// TwinCAT 3 PLC project lfe_motion
// Title: lcls-plc-lfe-motion
// Company: SLAC - LCLS
// ProjectVersion: 0.0.0
// ProgramVersion: 3.1.4026.17
// CompilerDefines: L
// libraries:
//   LCLS General, * (SLAC)
//   lcls-twincat-common-components, * (SLAC)
//   lcls-twincat-motion, * (SLAC)
//   lcls-twincat-physics, * (SLAC)
//   PMPS, * (SLAC - LCLS)
//   Tc2_MC2, * (Beckhoff Automation GmbH)
//   Tc2_SerialCom, * (Beckhoff Automation GmbH)
//   Tc2_Standard, * (Beckhoff Automation GmbH)
//   Tc2_System, * (Beckhoff Automation GmbH)
//   Tc3_Module, * (Beckhoff Automation GmbH)
// project tree:
//   DUTs/ DUT_SATT_Filter.TcDUT (not stored), ST_MPA.TcDUT (not stored), E_PositionState.TcDUT (not stored)
//   GVLs/ GVL.TcGVL, Main.TcGVL, RTDSL0.TcGVL (not stored)
//   / PlcTask.TcTTO
//   POUs/ FB_AttenuatorElementDensity.TcPOU (not stored), PRG_AL1L0_REF.TcPOU, PRG_IM5L0_PPM.TcPOU, PRG_3_PMPS_POST.TcPOU, PRG_4_LOG.TcPOU (not stored), PRG_AT2L0_SOLID.TcPOU, PRG_EM3L0_IPM.TcPOU, PRG_IM1L0_XTES.TcPOU, PRG_IM1L1_PPM.TcPOU (not stored), PRG_IM2L0_XTES.TcPOU, PRG_IM3L0_PPM.TcPOU, PRG_IM4L0_XTES.TcPOU, PRG_2_PMPS_PRE.TcPOU (not stored), PRG_1_PlcTask.TcPOU, PRG_RTDSL0.TcPOU (not stored), PRG_SL1L0_POWER.TcPOU (not stored), PRG_SL2L0_POWER.TcPOU (not stored), PRG_SL3L0_SCATTER.TcPOU, PRG_SP1L0_KMONO.TcPOU (not stored), PRG_PF1L0_WFS.TcPOU
//   Temp/ FB_AttFFO.TcPOU (not stored), FB_BasicAxisFFO.TcPOU (not stored), FB_BasicMotionStageAltFFO.TcPOU (not stored), FB_BasicMotionStageFFO.TcPOU (not stored), FB_MPA.TcPOU (not stored), FB_SimMotor.TcPOU (not stored), FB_SLITS.TcPOU (not stored), FB_SLITS_POWER.TcPOU (not stored), FB_SLITS_SCATTER.TcPOU
//   Version/ Global_Version.TcGVL
// real-time tasks:
//   TASK PlcTask: cycle T#10ms, priority 20, ADS port 350
// motion (NC):
//   TASK NC-Task 1 SAF: cycle T#1ms, priority 4, ADS port 501
//   TASK NC-Task 1 SVB: cycle T#10ms, priority 8, ADS port 511
//   AXIS Axis 1 (id 1)
//   AXIS Axis 2 (id 2)
//   AXIS Axis 3 (id 3)
//   AXIS Axis 4 (id 4)
//   AXIS Axis 5 (id 5)
//   AXIS Axis 6 (id 6)
//   AXIS Axis 7 (id 7)
//   AXIS Axis 8 (id 8)
//   AXIS Axis 9 (id 9)
//   AXIS Axis 10 (id 10)
//   AXIS Axis 11 (id 11)
//   AXIS Axis 12 (id 12)
//   AXIS Axis 13 (id 13)
//   AXIS Axis 14 (id 14)
//   AXIS Axis 15 (id 15)
//   AXIS Axis 16 (id 16)
//   AXIS Axis 17 (id 17)
//   AXIS Axis 18 (id 18)
//   AXIS Axis 19 (id 19)
//   AXIS Axis 20 IM1L0-XTES-MMS (id 20)
//   AXIS Axis 21 IM1L0-XTES-CLZ (id 21)
//   AXIS Axis 22 IM1L0-XTES-CLF (id 22)
//   AXIS Axis 23 IM1L1-PPM-MMS (id 23)
//   AXIS Axis 24 IM2L0-XTES-MMS (id 24)
//   AXIS Axis 25 IM2L0-XTES-CLZ (id 25)
//   AXIS Axis 26 IM2L0-XTES-CLF (id 26)
//   AXIS Axis 27 IM3L0-PPM-MMS (id 27)
//   AXIS Axis 28 IM4L0-XTES-MMS (id 28)
//   AXIS Axis 29 IM4L0-XTES-CLZ (id 29)
//   AXIS Axis 30 IM4L0-XTES-CLF (id 30)
//   AXIS PF1L0-WFS-MMS-01 (id 31)
//   AXIS PF1L0-WFS-MMS-02 (id 32)
//   AXIS Axis 33 (id 33)
//   AXIS Axis 34 (id 34)
//   AXIS Axis 35 (id 35)
//   AXIS Axis 36 (id 36)
//   AXIS Axis 37 (id 37)
//   AXIS Axis 38 (id 38)
//   AXIS Axis 39 (id 39)
//   AXIS Axis 40 (id 40)
//   AXIS SL1L0-BOTTOM-M41 (id 41)
//   AXIS SL1L0-SOUTH-M42 (id 42)
//   AXIS SL1L0-TOP-M43 (id 43)
//   AXIS SL1L0-NORTH-M44 (id 44)
//   AXIS SL2L0-BOTTOM-M45 (id 45)
//   AXIS SL2L0-SOUTH-M46 (id 46)
//   AXIS SL2L0-TOP-M47 (id 47)
//   AXIS SL2L0-NORTH-M48 (id 48)
//   AXIS XTAL ANGLE X (id 49)
//   AXIS XTAL VERT Y (id 50)
//   AXIS RETICLE HORIZ X (id 51)
//   AXIS RETICLE VERT Y (id 52)
//   AXIS DIODE HORIZ X (id 53)
//   AXIS DIODE VERT Y (id 54)
//   AXIS EM3L0-X-M55 (id 55)
//     Dynamic: AccelerationMaximum=50, DecelerationMaximum=50, Acceleration=50, Deceleration=50
//     Velo: RefSearch=0.1, RefSync=0.1, SlowManual=0.025, FastManual=0.05, Maximum=0.5
//     PositionAreaControl: Range=1
//     TargetPosControl: Range=0.001
//     OtherSettings: AllowMotionCmdToSlave=true
//     encoder EncType=29
//       EncPara: ScaleFactorNumerator=5e-05, Offset=-20.2296, MaxCount=#xffffffff, MaxCountHighDWord=#x0000001f
//         SoftEndMinControl: Enable=true, Range=-4
//         SoftEndMaxControl: Enable=true, Range=4
//         Inc: RefSoftSyncMask=#x0000ffff
//     drive DrvType=24
//       Analog: VeloReferenz=3.969, TorqueSetpointScale=10, ScaleFactorActTorque=0.1
//       TimeComp: TaskDelayCycles=1
//     controller CtrType=1
//       CtrPara: PriorControlFactor=1
//         PosDiffControl: Range=0.1
//         Observer: BandWidth=20
//   AXIS EM3L0-Y-M56 (id 56)
//     Dynamic: AccelerationMaximum=50, DecelerationMaximum=50, Acceleration=50, Deceleration=50
//     Velo: RefSearch=0.1, RefSync=0.1, SlowManual=0.025, FastManual=0.05, Maximum=2
//     PositionAreaControl: Enable=false
//     TargetPosControl: Range=0.025
//     OtherSettings: AllowMotionCmdToSlave=true
//     encoder EncType=29
//       EncPara: ScaleFactorNumerator=5e-05, Offset=3.65, Inverse=true, MaxCount=#xffffffff, MaxCountHighDWord=#x0000001f
//         SoftEndMinControl: Enable=true, Range=-81
//         SoftEndMaxControl: Enable=true, Range=1
//         Inc: RefSoftSyncMask=#x0000ffff
//     drive DrvType=24
//       Analog: VeloReferenz=12.5, TorqueSetpointScale=10, ScaleFactorActTorque=0.1
//       TimeComp: TaskDelayCycles=1
//     controller CtrType=1
//       CtrPara: PriorControlFactor=1
//         PosDiffControl: Enable=false, Range=0.03
//         Observer: BandWidth=20
//   AXIS Axis 57 IM5L0-PPM-MMS (id 57)
//     Dynamic: AccelerationMaximum=100, DecelerationMaximum=100, Acceleration=100, Deceleration=100, Jerk=1000
//     Velo: RefSearch=0.2, RefSync=0.2, SlowManual=0.05, FastManual=0.1, Maximum=1
//     TargetPosControl: Range=0.05
//     OtherSettings: AllowMotionCmdToSlave=true
//     encoder EncType=29
//       EncPara: ScaleFactorNumerator=5e-05, Offset=-6871886.7728, MaxCount=#xffffffff, MaxCountHighDWord=#x0000001f
//         SoftEndMinControl: Enable=true, Range=-105
//         SoftEndMaxControl: Enable=true
//         Inc: RefSoftSyncMask=#x0000ffff
//     drive DrvType=24
//       Analog: VeloReferenz=25, TorqueSetpointScale=10, ScaleFactorActTorque=0.1
//       TimeComp: TaskDelayCycles=1
//     controller CtrType=1
//       CtrPara: PriorControlFactor=1
//         PosDiffControl: Enable=false, Range=0.06
//         Observer: BandWidth=20
//   AXIS AL1L0-REF-MMS-M58 (id 58)
//     Dynamic: AccelerationMaximum=100, DecelerationMaximum=100, Acceleration=100, Deceleration=100
//     Velo: RefSearch=0.2, RefSync=0.2, SlowManual=0.05, FastManual=0.1, Maximum=1
//     PositionAreaControl: Range=1
//     TargetPosControl: Range=0.02
//     OtherSettings: AllowMotionCmdToSlave=true
//     encoder EncType=29
//       EncPara: ScaleFactorNumerator=5e-05, Offset=13.7558, Inverse=true, MaxCount=#xffffffff, MaxCountHighDWord=#x0000001f
//         SoftEndMinControl: Enable=true, Range=-47
//         SoftEndMaxControl: Enable=true, Range=2
//         Inc: RefSoftSyncMask=#x0000ffff
//     drive DrvType=24
//       Analog: VeloReferenz=5, TorqueSetpointScale=10, ScaleFactorActTorque=0.1
//       TimeComp: TaskDelayCycles=1
//     controller CtrType=1
//       CtrPara: PriorControlFactor=1
//         PosDiffControl: Range=1
//         PID: PosKp=2
//         Observer: BandWidth=20
//   AXIS SL3L0-BOTTOM-M59 (id 59)
//     Dynamic: AccelerationMaximum=100, DecelerationMaximum=100, Acceleration=100, Deceleration=100
//     Velo: Maximum=1
//     PositionAreaControl: Range=0.2
//     TargetPosControl: Range=0.005, Time=0.1
//     OtherSettings: AllowMotionCmdToSlave=true
//     encoder EncType=29
//       EncPara: ScaleFactorNumerator=5e-06, MaxCount=#xffffffff, MaxCountHighDWord=#x0000001f
//         SoftEndMinControl: Enable=true, Range=5.25
//         SoftEndMaxControl: Enable=true, Range=36.7
//         Inc: RefSoftSyncMask=#x0000ffff
//     drive DrvType=24
//       Analog: VeloReferenz=2, TorqueSetpointScale=10, ScaleFactorActTorque=0.1
//       TimeComp: TaskDelayCycles=1
//     controller CtrType=1
//       CtrPara: PriorControlFactor=1
//         PosDiffControl: Range=0.5
//         PID: PosKp=2
//         Observer: BandWidth=20
//   AXIS SL3L0-TOP-M60 (id 60)
//     Dynamic: AccelerationMaximum=100, DecelerationMaximum=100, Acceleration=100, Deceleration=100
//     Velo: Maximum=1
//     PositionAreaControl: Range=0.2
//     TargetPosControl: Range=0.005
//     OtherSettings: AllowMotionCmdToSlave=true
//     encoder EncType=29
//       EncPara: ScaleFactorNumerator=5e-06, MaxCount=#xffffffff, MaxCountHighDWord=#x0000001f
//         SoftEndMinControl: Enable=true, Range=4.5
//         SoftEndMaxControl: Enable=true, Range=33.3
//         Inc: RefSoftSyncMask=#x0000ffff
//     drive DrvType=24
//       Analog: VeloReferenz=2, TorqueSetpointScale=10, ScaleFactorActTorque=0.1
//       TimeComp: TaskDelayCycles=1
//     controller CtrType=1
//       CtrPara: PriorControlFactor=1
//         PosDiffControl: Range=0.5
//         PID: PosKp=2
//         Observer: BandWidth=20
//   AXIS SL3L0-SOUTH-M61 (id 61)
//     Dynamic: AccelerationMaximum=100, DecelerationMaximum=100, Acceleration=100, Deceleration=100
//     Velo: Maximum=1
//     PositionAreaControl: Range=0.2
//     TargetPosControl: Range=0.005
//     OtherSettings: AllowMotionCmdToSlave=true
//     encoder EncType=29
//       EncPara: ScaleFactorNumerator=5e-06, MaxCount=#xffffffff, MaxCountHighDWord=#x0000001f
//         SoftEndMinControl: Enable=true, Range=5
//         SoftEndMaxControl: Enable=true, Range=36.5
//         Inc: RefSoftSyncMask=#x0000ffff
//     drive DrvType=24
//       Analog: VeloReferenz=2, TorqueSetpointScale=10, ScaleFactorActTorque=0.1
//       TimeComp: TaskDelayCycles=1
//     controller CtrType=1
//       CtrPara: PriorControlFactor=1
//         PosDiffControl: Range=0.5
//         PID: PosKp=2
//         Observer: BandWidth=20
//   AXIS SL3L0-NORTH-M62 (id 62)
//     Dynamic: AccelerationMaximum=100, DecelerationMaximum=100, Acceleration=100, Deceleration=100
//     Velo: Maximum=1
//     PositionAreaControl: Range=0.2
//     TargetPosControl: Range=0.005
//     OtherSettings: AllowMotionCmdToSlave=true
//     encoder EncType=29
//       EncPara: ScaleFactorNumerator=5e-06, MaxCount=#xffffffff, MaxCountHighDWord=#x0000001f
//         SoftEndMinControl: Enable=true, Range=4.3
//         SoftEndMaxControl: Enable=true, Range=35.2
//         Inc: RefSoftSyncMask=#x0000ffff
//     drive DrvType=24
//       Analog: VeloReferenz=2, TorqueSetpointScale=10, ScaleFactorActTorque=0.1
//       TimeComp: TaskDelayCycles=1
//     controller CtrType=1
//       CtrPara: PriorControlFactor=1
//         PosDiffControl: Range=0.5
//         PID: PosKp=2
//         Observer: BandWidth=20
// I/O:
//   DEVICE PLC Rail (EtherCAT), AmsNetId 172.21.88.228.2.1
//     Power (EK1200) [EK1200-5000 EtherCAT Power supply (2A E-Bus)]
//       PMPS_FFO
//       License (EL6070)
//       PMPS_PRE
//       PLC Junction 1 (EK1122)
//       PLC Junction 2 (EK1122) [EK1122 2 port EtherCAT junction]
//         IM2L0 AT2L0 SL1L0 JUNCTION (CU1124)
//         X2 HXR EC2 (EK1100)
//         X2 SL2L0-Power (EK1100)
//       PLC Junction 3  (EK1122) [EK1122 2 port EtherCAT junction]
//         X1 B950-100H2-L0S5-ECJ-01 [CU1128 6x EtherCAT junction]
//           IM5L0-PPM [EK1100 EtherCAT Coupler (2A E-Bus)]
//             IM5L0-EL7047-E1 [EL7047 1Ch. Stepper motor output stage (50V, 5A)]
//             IM5L0-EL5042-E2 [EL5042 2Ch. BiSS-C Encoder]
//             IM5L0-EL2004-E3 [EL2004 4Ch. Dig. Output 24V, 0.5A]
//             IM5L0-EL1084-E4 [EL1084 4Ch. Dig. Input 24V, 3ms, negative]
//             IM5L0-EL3202-0010-E5 [EL3202-0010 2Ch. Ana. Input PT100 (RTD), High Precision]
//             IM5L0-EL3602-E6 [EL3602 2Ch. Ana. Input +/-10Volt, Diff. 24bit]
//             IM5L0-EL4004-E7 [EL4004 4Ch. Ana. Output 0-10V, 12bit]
//             IM5L0-EL2612-E8 [EL2612 2Ch. Relay Output, CO (125V AC / 30V DC)]
//             IM5L0-EL9011-E9 [EL9011 End Terminal]
//           SL3L0-SCATTER [EK1100 EtherCAT Coupler (2A E-Bus)]
//             SL3L0-EL7037-E1 [EL7037 1Ch. Stepper motor output stage (24V, 1.5A)]
//             SL3L0-EL5042-E2 [EL5042 2Ch. BiSS-C Encoder]
//             SL3L0-EL7037-E3 [EL7037 1Ch. Stepper motor output stage (24V, 1.5A)]
//             SL3L0-EL7037-E4 [EL7037 1Ch. Stepper motor output stage (24V, 1.5A)]
//             SL3L0-EL5042-E5 [EL5042 2Ch. BiSS-C Encoder]
//             SL3L0-EL7037-E6 [EL7037 1Ch. Stepper motor output stage (24V, 1.5A)]
//             SL3L0-EL9011-E7 [EL9011 End Terminal]
//           B950-100H2-L0S5-ECJ-01 (CU1128-B) [CU1128 6x EtherCAT junction - Dev A]
//             AL1L0-REF
//           B950-100H2-L0S5-ECJ-01 (CU1128-C) [CU1128 6x EtherCAT junction - Dev B]
// variable links:
//   (this object) <-> PLC Rail (EtherCAT)/Power (EK1200)/PLC Junction 2 (EK1122)/X2 HXR EC2 (EK1100)/EC2 E2 (EK1122)/X2 ECJ (CU1128)/X2 EM3L0-IPM (EK1100)/EM3L0-EL5042-E2
//     Enc/Inputs/In/nComState @bit 1 <-> WcState/InputToggle
//     Enc/Inputs/In/nComState <-> WcState/WcState
//     Enc/Inputs/In/nDataIn1 <-> FB Inputs Channel 1/Position
//     Enc/Inputs/In/nDataIn1 <-> FB Inputs Channel 2/Position
//     Enc/Inputs/In/nState1 @bit 12 <-> FB Inputs Channel 1/Status/Diag
//     Enc/Inputs/In/nState1 @bit 12 <-> FB Inputs Channel 2/Status/Diag
//     Enc/Inputs/In/nState1 @bit 1 <-> FB Inputs Channel 1/Status/Error
//     Enc/Inputs/In/nState1 @bit 1 <-> FB Inputs Channel 2/Status/Error
//     Enc/Inputs/In/nState1 @bit 14 <-> FB Inputs Channel 1/Status/Input cycle counter
//     Enc/Inputs/In/nState1 @bit 14 <-> FB Inputs Channel 2/Status/Input cycle counter
//     Enc/Inputs/In/nState1 @bit 2 <-> FB Inputs Channel 1/Status/Ready
//     Enc/Inputs/In/nState1 @bit 2 <-> FB Inputs Channel 2/Status/Ready
//     Enc/Inputs/In/nState1 @bit 13 <-> FB Inputs Channel 1/Status/TxPDO State
//     Enc/Inputs/In/nState1 @bit 13 <-> FB Inputs Channel 2/Status/TxPDO State
//     Enc/Inputs/In/nState1 <-> FB Inputs Channel 1/Status/Warning
//     Enc/Inputs/In/nState1 <-> FB Inputs Channel 2/Status/Warning
//   (this object) <-> PLC Rail (EtherCAT)/Power (EK1200)/PLC Junction 2 (EK1122)/X2 HXR EC2 (EK1100)/EC2 E2 (EK1122)/X2 ECJ (CU1128)/X2 EM3L0-IPM (EK1100)/EM3L0-EL7047-E1
//     Drive/Inputs/In/nState1 @bit 3 <-> STM Status/Status/Error
//     Drive/Inputs/In/nState1 @bit 7 <-> STM Status/Status/Motor stall
//     Drive/Inputs/In/nState1 @bit 5 <-> STM Status/Status/Moving negative
//     Drive/Inputs/In/nState1 @bit 4 <-> STM Status/Status/Moving positive
//     Drive/Inputs/In/nState1 @bit 1 <-> STM Status/Status/Ready
//     Drive/Inputs/In/nState1 <-> STM Status/Status/Ready to enable
//     Drive/Inputs/In/nState1 @bit 6 <-> STM Status/Status/Torque reduced
//     Drive/Inputs/In/nState1 @bit 2 <-> STM Status/Status/Warning
//     Drive/Inputs/In/nState2 @bit 3 <-> STM Status/Status/Digital input 1
//     Drive/Inputs/In/nState2 @bit 4 <-> STM Status/Status/Digital input 2
//     Drive/Inputs/In/nState2 @bit 5 <-> STM Status/Status/Sync error
//     Drive/Inputs/In/nState2 @bit 7 <-> STM Status/Status/TxPDO Toggle
//     Drive/Inputs/In/nState4 @bit 1 <-> WcState/InputToggle
//     Drive/Inputs/In/nState4 <-> WcState/WcState
//     Drive/Outputs/Out/nCtrl1 <-> STM Control/Control/Enable
//     Drive/Outputs/Out/nCtrl1 @bit 2 <-> STM Control/Control/Reduce torque
//     Drive/Outputs/Out/nCtrl1 @bit 1 <-> STM Control/Control/Reset
//     Drive/Outputs/Out/nCtrl2 @bit 3 <-> STM Control/Control/Digital output 1
//     Drive/Outputs/Out/nDataOut2[0] <-> STM Velocity/Velocity
//   (this object) <-> PLC Rail (EtherCAT)/Power (EK1200)/PLC Junction 2 (EK1122)/X2 HXR EC2 (EK1100)/EC2 E2 (EK1122)/X2 ECJ (CU1128)/X2 EM3L0-IPM (EK1100)/EM3L0-EL7047-E3
//     Drive/Inputs/In/nState1 @bit 3 <-> STM Status/Status/Error
//     Drive/Inputs/In/nState1 @bit 7 <-> STM Status/Status/Motor stall
//     Drive/Inputs/In/nState1 @bit 5 <-> STM Status/Status/Moving negative
//     Drive/Inputs/In/nState1 @bit 4 <-> STM Status/Status/Moving positive
//     Drive/Inputs/In/nState1 @bit 1 <-> STM Status/Status/Ready
//     Drive/Inputs/In/nState1 <-> STM Status/Status/Ready to enable
//     Drive/Inputs/In/nState1 @bit 6 <-> STM Status/Status/Torque reduced
//     Drive/Inputs/In/nState1 @bit 2 <-> STM Status/Status/Warning
//     Drive/Inputs/In/nState2 @bit 3 <-> STM Status/Status/Digital input 1
//     Drive/Inputs/In/nState2 @bit 4 <-> STM Status/Status/Digital input 2
//     Drive/Inputs/In/nState2 @bit 5 <-> STM Status/Status/Sync error
//     Drive/Inputs/In/nState2 @bit 7 <-> STM Status/Status/TxPDO Toggle
//     Drive/Inputs/In/nState4 @bit 1 <-> WcState/InputToggle
//     Drive/Inputs/In/nState4 <-> WcState/WcState
//     Drive/Outputs/Out/nCtrl1 <-> STM Control/Control/Enable
//     Drive/Outputs/Out/nCtrl1 @bit 2 <-> STM Control/Control/Reduce torque
//     Drive/Outputs/Out/nCtrl1 @bit 1 <-> STM Control/Control/Reset
//     Drive/Outputs/Out/nCtrl2 @bit 3 <-> STM Control/Control/Digital output 1
//     Drive/Outputs/Out/nDataOut2[0] <-> STM Velocity/Velocity
//   (this object) <-> PLC Rail (EtherCAT)/Power (EK1200)/PLC Junction 3  (EK1122)/X1 B950-100H2-L0S5-ECJ-01/IM5L0-PPM/IM5L0-EL5042-E2
//     Enc/Inputs/In/nComState @bit 1 <-> WcState/InputToggle
//     Enc/Inputs/In/nComState <-> WcState/WcState
//     Enc/Inputs/In/nDataIn1 <-> FB Inputs Channel 1/Position
//     Enc/Inputs/In/nState1 @bit 12 <-> FB Inputs Channel 1/Status/Diag
//     Enc/Inputs/In/nState1 @bit 1 <-> FB Inputs Channel 1/Status/Error
//     Enc/Inputs/In/nState1 @bit 14 <-> FB Inputs Channel 1/Status/Input cycle counter
//     Enc/Inputs/In/nState1 @bit 2 <-> FB Inputs Channel 1/Status/Ready
//     Enc/Inputs/In/nState1 @bit 13 <-> FB Inputs Channel 1/Status/TxPDO State
//     Enc/Inputs/In/nState1 <-> FB Inputs Channel 1/Status/Warning
//   (this object) <-> PLC Rail (EtherCAT)/Power (EK1200)/PLC Junction 3  (EK1122)/X1 B950-100H2-L0S5-ECJ-01/IM5L0-PPM/IM5L0-EL7047-E1
//     Drive/Inputs/In/nState1 @bit 3 <-> STM Status/Status/Error
//     Drive/Inputs/In/nState1 @bit 7 <-> STM Status/Status/Motor stall
//     Drive/Inputs/In/nState1 @bit 5 <-> STM Status/Status/Moving negative
//     Drive/Inputs/In/nState1 @bit 4 <-> STM Status/Status/Moving positive
//     Drive/Inputs/In/nState1 @bit 1 <-> STM Status/Status/Ready
//     Drive/Inputs/In/nState1 <-> STM Status/Status/Ready to enable
//     Drive/Inputs/In/nState1 @bit 6 <-> STM Status/Status/Torque reduced
//     Drive/Inputs/In/nState1 @bit 2 <-> STM Status/Status/Warning
//     Drive/Inputs/In/nState2 @bit 3 <-> STM Status/Status/Digital input 1
//     Drive/Inputs/In/nState2 @bit 4 <-> STM Status/Status/Digital input 2
//     Drive/Inputs/In/nState2 @bit 5 <-> STM Status/Status/Sync error
//     Drive/Inputs/In/nState2 @bit 7 <-> STM Status/Status/TxPDO Toggle
//     Drive/Inputs/In/nState4 @bit 1 <-> WcState/InputToggle
//     Drive/Inputs/In/nState4 <-> WcState/WcState
//     Drive/Outputs/Out/nCtrl1 <-> STM Control/Control/Enable
//     Drive/Outputs/Out/nCtrl1 @bit 2 <-> STM Control/Control/Reduce torque
//     Drive/Outputs/Out/nCtrl1 @bit 1 <-> STM Control/Control/Reset
//     Drive/Outputs/Out/nCtrl2 @bit 3 <-> STM Control/Control/Digital output 1
//     Drive/Outputs/Out/nDataOut2[0] <-> STM Velocity/Velocity
//   (this object) <-> PLC Rail (EtherCAT)/Power (EK1200)/PLC Junction 3  (EK1122)/X1 B950-100H2-L0S5-ECJ-01/B950-100H2-L0S5-ECJ-01 (CU1128-B)/AL1L0-REF/AL1L0-EL5042-E2
//     Enc/Inputs/In/nComState @bit 1 <-> WcState/InputToggle
//     Enc/Inputs/In/nComState <-> WcState/WcState
//     Enc/Inputs/In/nDataIn1 <-> FB Inputs Channel 2/Position
//     Enc/Inputs/In/nState1 @bit 12 <-> FB Inputs Channel 2/Status/Diag
//     Enc/Inputs/In/nState1 @bit 1 <-> FB Inputs Channel 2/Status/Error
//     Enc/Inputs/In/nState1 @bit 14 <-> FB Inputs Channel 2/Status/Input cycle counter
//     Enc/Inputs/In/nState1 @bit 2 <-> FB Inputs Channel 2/Status/Ready
//     Enc/Inputs/In/nState1 @bit 13 <-> FB Inputs Channel 2/Status/TxPDO State
//     Enc/Inputs/In/nState1 <-> FB Inputs Channel 2/Status/Warning
//   (this object) <-> PLC Rail (EtherCAT)/Power (EK1200)/PLC Junction 3  (EK1122)/X1 B950-100H2-L0S5-ECJ-01/B950-100H2-L0S5-ECJ-01 (CU1128-B)/AL1L0-REF/AL1L0-EL7047-E1
//     Drive/Inputs/In/nState1 @bit 3 <-> STM Status/Status/Error
//     Drive/Inputs/In/nState1 @bit 7 <-> STM Status/Status/Motor stall
//     Drive/Inputs/In/nState1 @bit 5 <-> STM Status/Status/Moving negative
//     Drive/Inputs/In/nState1 @bit 4 <-> STM Status/Status/Moving positive
//     Drive/Inputs/In/nState1 @bit 1 <-> STM Status/Status/Ready
//     Drive/Inputs/In/nState1 <-> STM Status/Status/Ready to enable
//     Drive/Inputs/In/nState1 @bit 6 <-> STM Status/Status/Torque reduced
//     Drive/Inputs/In/nState1 @bit 2 <-> STM Status/Status/Warning
//     Drive/Inputs/In/nState2 @bit 3 <-> STM Status/Status/Digital input 1
//     Drive/Inputs/In/nState2 @bit 4 <-> STM Status/Status/Digital input 2
//     Drive/Inputs/In/nState2 @bit 5 <-> STM Status/Status/Sync error
//     Drive/Inputs/In/nState2 @bit 7 <-> STM Status/Status/TxPDO Toggle
//     Drive/Inputs/In/nState4 @bit 1 <-> WcState/InputToggle
//     Drive/Inputs/In/nState4 <-> WcState/WcState
//     Drive/Outputs/Out/nCtrl1 <-> STM Control/Control/Enable
//     Drive/Outputs/Out/nCtrl1 @bit 2 <-> STM Control/Control/Reduce torque
//     Drive/Outputs/Out/nCtrl1 @bit 1 <-> STM Control/Control/Reset
//     Drive/Outputs/Out/nCtrl2 @bit 3 <-> STM Control/Control/Digital output 1
//     Drive/Outputs/Out/nDataOut2[0] <-> STM Velocity/Velocity
//   (this object) <-> PLC Rail (EtherCAT)/Power (EK1200)/PLC Junction 3  (EK1122)/X1 B950-100H2-L0S5-ECJ-01/SL3L0-SCATTER/SL3L0-EL5042-E5
//     Enc/Inputs/In/nComState @bit 1 <-> WcState/InputToggle
//     Enc/Inputs/In/nComState <-> WcState/WcState
//     Enc/Inputs/In/nDataIn1 <-> FB Inputs Channel 1/Position
//     Enc/Inputs/In/nDataIn1 <-> FB Inputs Channel 2/Position
//     Enc/Inputs/In/nState1 @bit 12 <-> FB Inputs Channel 1/Status/Diag
//     Enc/Inputs/In/nState1 @bit 12 <-> FB Inputs Channel 2/Status/Diag
//     Enc/Inputs/In/nState1 @bit 1 <-> FB Inputs Channel 1/Status/Error
//     Enc/Inputs/In/nState1 @bit 1 <-> FB Inputs Channel 2/Status/Error
//     Enc/Inputs/In/nState1 @bit 14 <-> FB Inputs Channel 1/Status/Input cycle counter
//     Enc/Inputs/In/nState1 @bit 14 <-> FB Inputs Channel 2/Status/Input cycle counter
//     Enc/Inputs/In/nState1 @bit 2 <-> FB Inputs Channel 1/Status/Ready
//     Enc/Inputs/In/nState1 @bit 2 <-> FB Inputs Channel 2/Status/Ready
//     Enc/Inputs/In/nState1 @bit 13 <-> FB Inputs Channel 1/Status/TxPDO State
//     Enc/Inputs/In/nState1 @bit 13 <-> FB Inputs Channel 2/Status/TxPDO State
//     Enc/Inputs/In/nState1 <-> FB Inputs Channel 1/Status/Warning
//     Enc/Inputs/In/nState1 <-> FB Inputs Channel 2/Status/Warning
//   (this object) <-> PLC Rail (EtherCAT)/Power (EK1200)/PLC Junction 3  (EK1122)/X1 B950-100H2-L0S5-ECJ-01/SL3L0-SCATTER/SL3L0-EL7037-E6
//     Drive/Inputs/In/nState1 @bit 3 <-> STM Status/Status/Error
//     Drive/Inputs/In/nState1 @bit 7 <-> STM Status/Status/Motor stall
//     Drive/Inputs/In/nState1 @bit 5 <-> STM Status/Status/Moving negative
//     Drive/Inputs/In/nState1 @bit 4 <-> STM Status/Status/Moving positive
//     Drive/Inputs/In/nState1 @bit 1 <-> STM Status/Status/Ready
//     Drive/Inputs/In/nState1 <-> STM Status/Status/Ready to enable
//     Drive/Inputs/In/nState1 @bit 6 <-> STM Status/Status/Torque reduced
//     Drive/Inputs/In/nState1 @bit 2 <-> STM Status/Status/Warning
//     Drive/Inputs/In/nState2 @bit 3 <-> STM Status/Status/Digital input 1
//     Drive/Inputs/In/nState2 @bit 4 <-> STM Status/Status/Digital input 2
//     Drive/Inputs/In/nState2 @bit 5 <-> STM Status/Status/Sync error
//     Drive/Inputs/In/nState2 @bit 7 <-> STM Status/Status/TxPDO Toggle
//     Drive/Inputs/In/nState4 @bit 1 <-> WcState/InputToggle
//     Drive/Inputs/In/nState4 <-> WcState/WcState
//     Drive/Outputs/Out/nCtrl1 <-> STM Control/Control/Enable
//     Drive/Outputs/Out/nCtrl1 @bit 2 <-> STM Control/Control/Reduce torque
//     Drive/Outputs/Out/nCtrl1 @bit 1 <-> STM Control/Control/Reset
//     Drive/Outputs/Out/nCtrl2 @bit 3 <-> STM Control/Control/Digital output 1
//     Drive/Outputs/Out/nDataOut2[0] <-> STM Velocity/Velocity
//   (this object) <-> PLC Rail (EtherCAT)/Power (EK1200)/PLC Junction 3  (EK1122)/X1 B950-100H2-L0S5-ECJ-01/SL3L0-SCATTER/SL3L0-EL7037-E4
//     Drive/Inputs/In/nState1 @bit 3 <-> STM Status/Status/Error
//     Drive/Inputs/In/nState1 @bit 7 <-> STM Status/Status/Motor stall
//     Drive/Inputs/In/nState1 @bit 5 <-> STM Status/Status/Moving negative
//     Drive/Inputs/In/nState1 @bit 4 <-> STM Status/Status/Moving positive
//     Drive/Inputs/In/nState1 @bit 1 <-> STM Status/Status/Ready
//     Drive/Inputs/In/nState1 <-> STM Status/Status/Ready to enable
//     Drive/Inputs/In/nState1 @bit 6 <-> STM Status/Status/Torque reduced
//     Drive/Inputs/In/nState1 @bit 2 <-> STM Status/Status/Warning
//     Drive/Inputs/In/nState2 @bit 3 <-> STM Status/Status/Digital input 1
//     Drive/Inputs/In/nState2 @bit 4 <-> STM Status/Status/Digital input 2
//     Drive/Inputs/In/nState2 @bit 5 <-> STM Status/Status/Sync error
//     Drive/Inputs/In/nState2 @bit 7 <-> STM Status/Status/TxPDO Toggle
//     Drive/Inputs/In/nState4 @bit 1 <-> WcState/InputToggle
//     Drive/Inputs/In/nState4 <-> WcState/WcState
//     Drive/Outputs/Out/nCtrl1 <-> STM Control/Control/Enable
//     Drive/Outputs/Out/nCtrl1 @bit 2 <-> STM Control/Control/Reduce torque
//     Drive/Outputs/Out/nCtrl1 @bit 1 <-> STM Control/Control/Reset
//     Drive/Outputs/Out/nCtrl2 @bit 3 <-> STM Control/Control/Digital output 1
//     Drive/Outputs/Out/nDataOut2[0] <-> STM Velocity/Velocity
//   (this object) <-> PLC Rail (EtherCAT)/Power (EK1200)/PLC Junction 3  (EK1122)/X1 B950-100H2-L0S5-ECJ-01/SL3L0-SCATTER/SL3L0-EL5042-E2
//     Enc/Inputs/In/nComState @bit 1 <-> WcState/InputToggle
//     Enc/Inputs/In/nComState <-> WcState/WcState
//     Enc/Inputs/In/nDataIn1 <-> FB Inputs Channel 1/Position
//     Enc/Inputs/In/nDataIn1 <-> FB Inputs Channel 2/Position
//     Enc/Inputs/In/nState1 @bit 12 <-> FB Inputs Channel 1/Status/Diag
//     Enc/Inputs/In/nState1 @bit 12 <-> FB Inputs Channel 2/Status/Diag
//     Enc/Inputs/In/nState1 @bit 1 <-> FB Inputs Channel 1/Status/Error
//     Enc/Inputs/In/nState1 @bit 1 <-> FB Inputs Channel 2/Status/Error
//     Enc/Inputs/In/nState1 @bit 14 <-> FB Inputs Channel 1/Status/Input cycle counter
//     Enc/Inputs/In/nState1 @bit 14 <-> FB Inputs Channel 2/Status/Input cycle counter
//     Enc/Inputs/In/nState1 @bit 2 <-> FB Inputs Channel 1/Status/Ready
//     Enc/Inputs/In/nState1 @bit 2 <-> FB Inputs Channel 2/Status/Ready
//     Enc/Inputs/In/nState1 @bit 13 <-> FB Inputs Channel 1/Status/TxPDO State
//     Enc/Inputs/In/nState1 @bit 13 <-> FB Inputs Channel 2/Status/TxPDO State
//     Enc/Inputs/In/nState1 <-> FB Inputs Channel 1/Status/Warning
//     Enc/Inputs/In/nState1 <-> FB Inputs Channel 2/Status/Warning
//   (this object) <-> PLC Rail (EtherCAT)/Power (EK1200)/PLC Junction 3  (EK1122)/X1 B950-100H2-L0S5-ECJ-01/SL3L0-SCATTER/SL3L0-EL7037-E3
//     Drive/Inputs/In/nState1 @bit 3 <-> STM Status/Status/Error
//     Drive/Inputs/In/nState1 @bit 7 <-> STM Status/Status/Motor stall
//     Drive/Inputs/In/nState1 @bit 5 <-> STM Status/Status/Moving negative
//     Drive/Inputs/In/nState1 @bit 4 <-> STM Status/Status/Moving positive
//     Drive/Inputs/In/nState1 @bit 1 <-> STM Status/Status/Ready
//     Drive/Inputs/In/nState1 <-> STM Status/Status/Ready to enable
//     Drive/Inputs/In/nState1 @bit 6 <-> STM Status/Status/Torque reduced
//     Drive/Inputs/In/nState1 @bit 2 <-> STM Status/Status/Warning
//     Drive/Inputs/In/nState2 @bit 3 <-> STM Status/Status/Digital input 1
//     Drive/Inputs/In/nState2 @bit 4 <-> STM Status/Status/Digital input 2
//     Drive/Inputs/In/nState2 @bit 5 <-> STM Status/Status/Sync error
//     Drive/Inputs/In/nState2 @bit 7 <-> STM Status/Status/TxPDO Toggle
//     Drive/Inputs/In/nState4 @bit 1 <-> WcState/InputToggle
//     Drive/Inputs/In/nState4 <-> WcState/WcState
//     Drive/Outputs/Out/nCtrl1 <-> STM Control/Control/Enable
//     Drive/Outputs/Out/nCtrl1 @bit 2 <-> STM Control/Control/Reduce torque
//     Drive/Outputs/Out/nCtrl1 @bit 1 <-> STM Control/Control/Reset
//     Drive/Outputs/Out/nCtrl2 @bit 3 <-> STM Control/Control/Digital output 1
//     Drive/Outputs/Out/nDataOut2[0] <-> STM Velocity/Velocity
//   (this object) <-> PLC Rail (EtherCAT)/Power (EK1200)/PLC Junction 3  (EK1122)/X1 B950-100H2-L0S5-ECJ-01/SL3L0-SCATTER/SL3L0-EL7037-E1
//     Drive/Inputs/In/nState1 @bit 3 <-> STM Status/Status/Error
//     Drive/Inputs/In/nState1 @bit 7 <-> STM Status/Status/Motor stall
//     Drive/Inputs/In/nState1 @bit 5 <-> STM Status/Status/Moving negative
//     Drive/Inputs/In/nState1 @bit 4 <-> STM Status/Status/Moving positive
//     Drive/Inputs/In/nState1 @bit 1 <-> STM Status/Status/Ready
//     Drive/Inputs/In/nState1 <-> STM Status/Status/Ready to enable
//     Drive/Inputs/In/nState1 @bit 6 <-> STM Status/Status/Torque reduced
//     Drive/Inputs/In/nState1 @bit 2 <-> STM Status/Status/Warning
//     Drive/Inputs/In/nState2 @bit 3 <-> STM Status/Status/Digital input 1
//     Drive/Inputs/In/nState2 @bit 4 <-> STM Status/Status/Digital input 2
//     Drive/Inputs/In/nState2 @bit 5 <-> STM Status/Status/Sync error
//     Drive/Inputs/In/nState2 @bit 7 <-> STM Status/Status/TxPDO Toggle
//     Drive/Inputs/In/nState4 @bit 1 <-> WcState/InputToggle
//     Drive/Inputs/In/nState4 <-> WcState/WcState
//     Drive/Outputs/Out/nCtrl1 <-> STM Control/Control/Enable
//     Drive/Outputs/Out/nCtrl1 @bit 2 <-> STM Control/Control/Reduce torque
//     Drive/Outputs/Out/nCtrl1 @bit 1 <-> STM Control/Control/Reset
//     Drive/Outputs/Out/nCtrl2 @bit 3 <-> STM Control/Control/Digital output 1
//     Drive/Outputs/Out/nDataOut2[0] <-> STM Velocity/Velocity
//   lfe_motion Instance <-> PLC Rail (EtherCAT)/Power (EK1200)/PLC Junction 1 (EK1122)/X1 RTDSL0 (EK1100)/RTDSL0-EL7041-01
//     PlcTask Inputs/Main.M33.bLimitBackwardEnable <-> STM Status/Status/Digital input 2
//     PlcTask Inputs/Main.M33.bLimitForwardEnable <-> STM Status/Status/Digital input 1
//   lfe_motion Instance <-> PLC Rail (EtherCAT)/Power (EK1200)/PLC Junction 1 (EK1122)/X1 RTDSL0 (EK1100)/RTDSL0-EL7041-05
//     PlcTask Inputs/Main.M38.bLimitBackwardEnable <-> STM Status/Status/Digital input 2
//     PlcTask Inputs/Main.M38.bLimitForwardEnable <-> STM Status/Status/Digital input 1
//   lfe_motion Instance <-> PLC Rail (EtherCAT)/Power (EK1200)/PLC Junction 1 (EK1122)/X1 RTDSL0 (EK1100)/RTDSL0-MPA-EL1008
//     PlcTask Inputs/RTDSL0.RTDSL0_MPA_01.i_xInsertedLS <-> Channel 1/Input
//     PlcTask Inputs/RTDSL0.RTDSL0_MPA_02.i_xInsertedLS <-> Channel 3/Input
//     PlcTask Inputs/RTDSL0.RTDSL0_MPA_03.i_xInsertedLS <-> Channel 5/Input
//     PlcTask Inputs/RTDSL0.RTDSL0_MPA_04.i_xInsertedLS <-> Channel 7/Input
//     PlcTask Inputs/RTDSL0.RTDSL0_MPA_01.i_xRetractedLS <-> Channel 2/Input
//     PlcTask Inputs/RTDSL0.RTDSL0_MPA_02.i_xRetractedLS <-> Channel 4/Input
//     PlcTask Inputs/RTDSL0.RTDSL0_MPA_03.i_xRetractedLS <-> Channel 6/Input
//     PlcTask Inputs/RTDSL0.RTDSL0_MPA_04.i_xRetractedLS <-> Channel 8/Input
//   lfe_motion Instance <-> PLC Rail (EtherCAT)/Power (EK1200)/PLC Junction 1 (EK1122)/X1 RTDSL0 (EK1100)/RTDSL0-MPA-EL2008
//     PlcTask Outputs/RTDSL0.RTDSL0_MPA_01.q_xInsert_DO <-> Channel 1/Output
//     PlcTask Outputs/RTDSL0.RTDSL0_MPA_02.q_xInsert_DO <-> Channel 3/Output
//     PlcTask Outputs/RTDSL0.RTDSL0_MPA_03.q_xInsert_DO <-> Channel 5/Output
//     PlcTask Outputs/RTDSL0.RTDSL0_MPA_04.q_xInsert_DO <-> Channel 7/Output
//     PlcTask Outputs/RTDSL0.RTDSL0_MPA_01.q_xRetract_DO <-> Channel 2/Output
//     PlcTask Outputs/RTDSL0.RTDSL0_MPA_02.q_xRetract_DO <-> Channel 4/Output
//     PlcTask Outputs/RTDSL0.RTDSL0_MPA_03.q_xRetract_DO <-> Channel 6/Output
//     PlcTask Outputs/RTDSL0.RTDSL0_MPA_04.q_xRetract_DO <-> Channel 8/Output
//   lfe_motion Instance <-> PLC Rail (EtherCAT)/Power (EK1200)/PLC Junction 1 (EK1122)/X1 RTDSL0 (EK1100)/Term 113 (EL3054)
//     PlcTask Inputs/Main.M38.nRawEncoderINT <-> AI Standard Channel 1/Value
//   lfe_motion Instance <-> PLC Rail (EtherCAT)/Power (EK1200)/PLC Junction 1 (EK1122)/X2 IM1L0-XTES (EK1100)/IM1L0-EL1088
//     PlcTask Inputs/Main.M21.bHome <-> Channel 2/Input
//     PlcTask Inputs/Main.M22.bHome <-> Channel 4/Input
//     PlcTask Inputs/PRG_IM1L0_XTES.fbIM1L0.bFocusEndBwd <-> Channel 4/Input
//     PlcTask Inputs/PRG_IM1L0_XTES.fbIM1L0.bFocusEndFwd <-> Channel 3/Input
//     PlcTask Inputs/PRG_IM1L0_XTES.fbIM1L0.bZoomEndBwd <-> Channel 2/Input
//     PlcTask Inputs/PRG_IM1L0_XTES.fbIM1L0.bZoomEndFwd <-> Channel 1/Input
//   lfe_motion Instance <-> PLC Rail (EtherCAT)/Power (EK1200)/PLC Junction 1 (EK1122)/X2 IM1L0-XTES (EK1100)/IM1L0-EL2004
//     PlcTask Outputs/Main.M20.bBrakeRelease <-> Channel 1/Output
//     PlcTask Outputs/PRG_IM1L0_XTES.fbIM1L0.fbLED.bLEDPower <-> Channel 3/Output
//     PlcTask Outputs/PRG_IM1L0_XTES.fbIM1L0.fbOpal.bOpalPower <-> Channel 2/Output
//   lfe_motion Instance <-> PLC Rail (EtherCAT)/Power (EK1200)/PLC Junction 1 (EK1122)/X2 IM1L0-XTES (EK1100)/IM1L0-EL6002
//     PlcTask Inputs/PRG_IM1L0_XTES.stEL6In/D[{0..21}] <-> COM TxPDO-Map Inputs Channel 1/Data In {0..21}  (22 links)
//     PlcTask Inputs/PRG_IM1L0_XTES.stEL6In/Status <-> COM TxPDO-Map Inputs Channel 1/Status
//     PlcTask Outputs/PRG_IM1L0_XTES.stEL6Out/Ctrl <-> COM RxPDO-Map Outputs Channel 1/Ctrl
//     PlcTask Outputs/PRG_IM1L0_XTES.stEL6Out/D[{0..21}] <-> COM RxPDO-Map Outputs Channel 1/Data Out {0..21}  (22 links)
//   lfe_motion Instance <-> PLC Rail (EtherCAT)/Power (EK1200)/PLC Junction 1 (EK1122)/X2 IM1L0-XTES (EK1100)/IM1L0-EL7041
//     PlcTask Inputs/Main.M20.bLimitForwardEnable <-> STM Status/Status/Digital input 1
//   lfe_motion Instance <-> PLC Rail (EtherCAT)/Power (EK1200)/PLC Junction 1 (EK1122)/X2 IM1L0-XTES (EK1100)/IM1L0-EL7342
//     PlcTask Inputs/PRG_IM1L0_XTES.bIM1L0FlowOk <-> DCM Status Channel 1/Status/Digital input 1
//   lfe_motion Instance <-> PLC Rail (EtherCAT)/Power (EK1200)/PLC Junction 2 (EK1122)/IM2L0 AT2L0 SL1L0 JUNCTION (CU1124)/X1 IM2L0-XTES (EK1100)/IM2L0-EL1088
//     PlcTask Inputs/Main.M25.bHome <-> Channel 2/Input
//     PlcTask Inputs/Main.M26.bHome <-> Channel 4/Input
//     PlcTask Inputs/PRG_IM2L0_XTES.fbIM2L0.bFocusEndBwd <-> Channel 4/Input
//     PlcTask Inputs/PRG_IM2L0_XTES.fbIM2L0.bFocusEndFwd <-> Channel 3/Input
//     PlcTask Inputs/PRG_IM2L0_XTES.fbIM2L0.bZoomEndBwd <-> Channel 2/Input
//     PlcTask Inputs/PRG_IM2L0_XTES.fbIM2L0.bZoomEndFwd <-> Channel 1/Input
//   lfe_motion Instance <-> PLC Rail (EtherCAT)/Power (EK1200)/PLC Junction 2 (EK1122)/IM2L0 AT2L0 SL1L0 JUNCTION (CU1124)/X1 IM2L0-XTES (EK1100)/IM2L0-EL2004
//     PlcTask Outputs/Main.M24.bBrakeRelease <-> Channel 1/Output
//     PlcTask Outputs/PRG_IM2L0_XTES.fbIM2L0.fbLED.bLEDPower <-> Channel 3/Output
//     PlcTask Outputs/PRG_IM2L0_XTES.fbIM2L0.fbOpal.bOpalPower <-> Channel 2/Output
//   lfe_motion Instance <-> PLC Rail (EtherCAT)/Power (EK1200)/PLC Junction 2 (EK1122)/IM2L0 AT2L0 SL1L0 JUNCTION (CU1124)/X1 IM2L0-XTES (EK1100)/IM2L0-EL6002
//     PlcTask Inputs/PRG_IM2L0_XTES.stEL6In/D[{0..21}] <-> COM TxPDO-Map Inputs Channel 1/Data In {0..21}  (22 links)
//     PlcTask Inputs/PRG_IM2L0_XTES.stEL6In/Status <-> COM TxPDO-Map Inputs Channel 1/Status
//     PlcTask Outputs/PRG_IM2L0_XTES.stEL6Out/Ctrl <-> COM RxPDO-Map Outputs Channel 1/Ctrl
//     PlcTask Outputs/PRG_IM2L0_XTES.stEL6Out/D[{0..21}] <-> COM RxPDO-Map Outputs Channel 1/Data Out {0..21}  (22 links)
//   lfe_motion Instance <-> PLC Rail (EtherCAT)/Power (EK1200)/PLC Junction 2 (EK1122)/IM2L0 AT2L0 SL1L0 JUNCTION (CU1124)/X1 IM2L0-XTES (EK1100)/IM2L0-EL7041
//     PlcTask Inputs/PRG_IM2L0_XTES.bDefectiveLimitSwitch <-> STM Status/Status/Digital input 1
//   lfe_motion Instance <-> PLC Rail (EtherCAT)/Power (EK1200)/PLC Junction 2 (EK1122)/IM2L0 AT2L0 SL1L0 JUNCTION (CU1124)/X1 PF1L0-WFS (EK1100)/PF1L0-EL2004
//     PlcTask Outputs/Main.M31.bBrakeRelease <-> Channel 1/Output
//   lfe_motion Instance <-> PLC Rail (EtherCAT)/Power (EK1200)/PLC Junction 2 (EK1122)/IM2L0 AT2L0 SL1L0 JUNCTION (CU1124)/X1 PF1L0-WFS (EK1100)/PF1L0-EL3314
//     PlcTask Inputs/PRG_PF1L0_WFS.fbPF1L0.fbThermoCouple1.bError <-> TC Inputs Channel 1/Status/Error
//     PlcTask Inputs/PRG_PF1L0_WFS.fbPF1L0.fbThermoCouple2.bError <-> TC Inputs Channel 2/Status/Error
//     PlcTask Inputs/PRG_PF1L0_WFS.fbPF1L0.fbThermoCouple1.bOverrange <-> TC Inputs Channel 1/Status/Overrange
//     PlcTask Inputs/PRG_PF1L0_WFS.fbPF1L0.fbThermoCouple2.bOverrange <-> TC Inputs Channel 2/Status/Overrange
//     PlcTask Inputs/PRG_PF1L0_WFS.fbPF1L0.fbThermoCouple1.bUnderrange <-> TC Inputs Channel 1/Status/Underrange
//     PlcTask Inputs/PRG_PF1L0_WFS.fbPF1L0.fbThermoCouple2.bUnderrange <-> TC Inputs Channel 2/Status/Underrange
//     PlcTask Inputs/PRG_PF1L0_WFS.fbPF1L0.fbThermoCouple1.iRaw <-> TC Inputs Channel 1/Value
//     PlcTask Inputs/PRG_PF1L0_WFS.fbPF1L0.fbThermoCouple2.iRaw <-> TC Inputs Channel 2/Value
//   lfe_motion Instance <-> PLC Rail (EtherCAT)/Power (EK1200)/PLC Junction 2 (EK1122)/IM2L0 AT2L0 SL1L0 JUNCTION (CU1124)/X1 PF1L0-WFS (EK1100)/PF1L0-EL5042
//     PlcTask Inputs/Main.M31.nRawEncoderULINT <-> FB Inputs Channel 2/Position
//     PlcTask Inputs/Main.M32.nRawEncoderULINT <-> FB Inputs Channel 1/Position
//   lfe_motion Instance <-> PLC Rail (EtherCAT)/Power (EK1200)/PLC Junction 2 (EK1122)/IM2L0 AT2L0 SL1L0 JUNCTION (CU1124)/X1 PF1L0-WFS (EK1100)/PF1L0-EL7041-01
//     PlcTask Inputs/Main.M31.bLimitBackwardEnable <-> STM Status/Status/Digital input 2
//     PlcTask Inputs/Main.M31.bLimitForwardEnable <-> STM Status/Status/Digital input 1
//   lfe_motion Instance <-> PLC Rail (EtherCAT)/Power (EK1200)/PLC Junction 2 (EK1122)/IM2L0 AT2L0 SL1L0 JUNCTION (CU1124)/X1 SL1L0-Power (EK1100)/SL1L0-EL3202-E10
//     PlcTask Inputs/PRG_SL1L0_POWER.fbSL1L0.RTD_TOP_1.bError <-> RTD Inputs Channel 1/Status/Error
//     PlcTask Inputs/PRG_SL1L0_POWER.fbSL1L0.RTD_TOP_2.bError <-> RTD Inputs Channel 2/Status/Error
//     PlcTask Inputs/PRG_SL1L0_POWER.fbSL1L0.RTD_TOP_1.bOverrange <-> RTD Inputs Channel 1/Status/Overrange
//     PlcTask Inputs/PRG_SL1L0_POWER.fbSL1L0.RTD_TOP_2.bOverrange <-> RTD Inputs Channel 2/Status/Overrange
//     PlcTask Inputs/PRG_SL1L0_POWER.fbSL1L0.RTD_TOP_1.bUnderrange <-> RTD Inputs Channel 1/Status/Underrange
//     PlcTask Inputs/PRG_SL1L0_POWER.fbSL1L0.RTD_TOP_2.bUnderrange <-> RTD Inputs Channel 2/Status/Underrange
//     PlcTask Inputs/PRG_SL1L0_POWER.fbSL1L0.RTD_TOP_1.iRaw <-> RTD Inputs Channel 1/Value
//     PlcTask Inputs/PRG_SL1L0_POWER.fbSL1L0.RTD_TOP_2.iRaw <-> RTD Inputs Channel 2/Value
//   lfe_motion Instance <-> PLC Rail (EtherCAT)/Power (EK1200)/PLC Junction 2 (EK1122)/IM2L0 AT2L0 SL1L0 JUNCTION (CU1124)/X1 SL1L0-Power (EK1100)/SL1L0-EL3202-E11
//     PlcTask Inputs/PRG_SL1L0_POWER.fbSL1L0.RTD_North_1.bError <-> RTD Inputs Channel 1/Status/Error
//     PlcTask Inputs/PRG_SL1L0_POWER.fbSL1L0.RTD_North_2.bError <-> RTD Inputs Channel 2/Status/Error
//     PlcTask Inputs/PRG_SL1L0_POWER.fbSL1L0.RTD_North_1.bOverrange <-> RTD Inputs Channel 1/Status/Overrange
//     PlcTask Inputs/PRG_SL1L0_POWER.fbSL1L0.RTD_North_2.bOverrange <-> RTD Inputs Channel 2/Status/Overrange
//     PlcTask Inputs/PRG_SL1L0_POWER.fbSL1L0.RTD_North_1.bUnderrange <-> RTD Inputs Channel 1/Status/Underrange
//     PlcTask Inputs/PRG_SL1L0_POWER.fbSL1L0.RTD_North_2.bUnderrange <-> RTD Inputs Channel 2/Status/Underrange
//     PlcTask Inputs/PRG_SL1L0_POWER.fbSL1L0.RTD_North_1.iRaw <-> RTD Inputs Channel 1/Value
//     PlcTask Inputs/PRG_SL1L0_POWER.fbSL1L0.RTD_North_2.iRaw <-> RTD Inputs Channel 2/Value
//   lfe_motion Instance <-> PLC Rail (EtherCAT)/Power (EK1200)/PLC Junction 2 (EK1122)/IM2L0 AT2L0 SL1L0 JUNCTION (CU1124)/X1 SL1L0-Power (EK1100)/SL1L0-EL3202-E8
//     PlcTask Inputs/PRG_SL1L0_POWER.fbSL1L0.RTD_Bottom_1.bError <-> RTD Inputs Channel 1/Status/Error
//     PlcTask Inputs/PRG_SL1L0_POWER.fbSL1L0.RTD_Bottom_2.bError <-> RTD Inputs Channel 2/Status/Error
//     PlcTask Inputs/PRG_SL1L0_POWER.fbSL1L0.RTD_Bottom_1.bOverrange <-> RTD Inputs Channel 1/Status/Overrange
//     PlcTask Inputs/PRG_SL1L0_POWER.fbSL1L0.RTD_Bottom_2.bOverrange <-> RTD Inputs Channel 2/Status/Overrange
//     PlcTask Inputs/PRG_SL1L0_POWER.fbSL1L0.RTD_Bottom_1.bUnderrange <-> RTD Inputs Channel 1/Status/Underrange
//     PlcTask Inputs/PRG_SL1L0_POWER.fbSL1L0.RTD_Bottom_2.bUnderrange <-> RTD Inputs Channel 2/Status/Underrange
//     PlcTask Inputs/PRG_SL1L0_POWER.fbSL1L0.RTD_Bottom_1.iRaw <-> RTD Inputs Channel 1/Value
//     PlcTask Inputs/PRG_SL1L0_POWER.fbSL1L0.RTD_Bottom_2.iRaw <-> RTD Inputs Channel 2/Value
//   lfe_motion Instance <-> PLC Rail (EtherCAT)/Power (EK1200)/PLC Junction 2 (EK1122)/IM2L0 AT2L0 SL1L0 JUNCTION (CU1124)/X1 SL1L0-Power (EK1100)/SL1L0-EL3202-E9
//     PlcTask Inputs/PRG_SL1L0_POWER.fbSL1L0.RTD_South_1.bError <-> RTD Inputs Channel 1/Status/Error
//     PlcTask Inputs/PRG_SL1L0_POWER.fbSL1L0.RTD_South_2.bError <-> RTD Inputs Channel 2/Status/Error
//     PlcTask Inputs/PRG_SL1L0_POWER.fbSL1L0.RTD_South_1.bOverrange <-> RTD Inputs Channel 1/Status/Overrange
//     PlcTask Inputs/PRG_SL1L0_POWER.fbSL1L0.RTD_South_2.bOverrange <-> RTD Inputs Channel 2/Status/Overrange
//     PlcTask Inputs/PRG_SL1L0_POWER.fbSL1L0.RTD_South_1.bUnderrange <-> RTD Inputs Channel 1/Status/Underrange
//     PlcTask Inputs/PRG_SL1L0_POWER.fbSL1L0.RTD_South_2.bUnderrange <-> RTD Inputs Channel 2/Status/Underrange
//     PlcTask Inputs/PRG_SL1L0_POWER.fbSL1L0.RTD_South_1.iRaw <-> RTD Inputs Channel 1/Value
//     PlcTask Inputs/PRG_SL1L0_POWER.fbSL1L0.RTD_South_2.iRaw <-> RTD Inputs Channel 2/Value
//   lfe_motion Instance <-> PLC Rail (EtherCAT)/Power (EK1200)/PLC Junction 2 (EK1122)/IM2L0 AT2L0 SL1L0 JUNCTION (CU1124)/X1 SL1L0-Power (EK1100)/SL1L0-EL7041-E1
//     PlcTask Inputs/Main.M41.bLimitBackwardEnable <-> STM Status/Status/Digital input 1
//     PlcTask Inputs/Main.M41.bLimitForwardEnable <-> STM Status/Status/Digital input 2
//   lfe_motion Instance <-> PLC Rail (EtherCAT)/Power (EK1200)/PLC Junction 2 (EK1122)/IM2L0 AT2L0 SL1L0 JUNCTION (CU1124)/X1 SL1L0-Power (EK1100)/SL1L0-EL7041-E3
//     PlcTask Inputs/Main.M42.bLimitBackwardEnable <-> STM Status/Status/Digital input 2
//     PlcTask Inputs/Main.M42.bLimitForwardEnable <-> STM Status/Status/Digital input 1
//   lfe_motion Instance <-> PLC Rail (EtherCAT)/Power (EK1200)/PLC Junction 2 (EK1122)/IM2L0 AT2L0 SL1L0 JUNCTION (CU1124)/X1 SL1L0-Power (EK1100)/SL1L0-EL7041-E5
//     PlcTask Inputs/Main.M43.bLimitBackwardEnable <-> STM Status/Status/Digital input 1
//     PlcTask Inputs/Main.M43.bLimitForwardEnable <-> STM Status/Status/Digital input 2
//   lfe_motion Instance <-> PLC Rail (EtherCAT)/Power (EK1200)/PLC Junction 2 (EK1122)/IM2L0 AT2L0 SL1L0 JUNCTION (CU1124)/X1 SL1L0-Power (EK1100)/SL1L0-EL7041-E7
//     PlcTask Inputs/Main.M44.bLimitBackwardEnable <-> STM Status/Status/Digital input 2
//     PlcTask Inputs/Main.M44.bLimitForwardEnable <-> STM Status/Status/Digital input 1
//   lfe_motion Instance <-> PLC Rail (EtherCAT)/Power (EK1200)/PLC Junction 2 (EK1122)/IM2L0 AT2L0 SL1L0 JUNCTION (CU1124)/X2 AT2L0-SOLID (EK1100)/AT2L0-EL7041-01
//     PlcTask Inputs/Main.M1.bLimitBackwardEnable <-> STM Status/Status/Digital input 1
//     PlcTask Inputs/Main.M1.bLimitForwardEnable <-> STM Status/Status/Digital input 2
//   lfe_motion Instance <-> PLC Rail (EtherCAT)/Power (EK1200)/PLC Junction 2 (EK1122)/IM2L0 AT2L0 SL1L0 JUNCTION (CU1124)/X2 AT2L0-SOLID (EK1100)/AT2L0-EL7041-02
//     PlcTask Inputs/Main.M2.bLimitBackwardEnable <-> STM Status/Status/Digital input 1
//     PlcTask Inputs/Main.M2.bLimitForwardEnable <-> STM Status/Status/Digital input 2
//   lfe_motion Instance <-> PLC Rail (EtherCAT)/Power (EK1200)/PLC Junction 2 (EK1122)/IM2L0 AT2L0 SL1L0 JUNCTION (CU1124)/X2 AT2L0-SOLID (EK1100)/AT2L0-EL7041-03
//     PlcTask Inputs/Main.M3.bLimitBackwardEnable <-> STM Status/Status/Digital input 1
//     PlcTask Inputs/Main.M3.bLimitForwardEnable <-> STM Status/Status/Digital input 2
//   lfe_motion Instance <-> PLC Rail (EtherCAT)/Power (EK1200)/PLC Junction 2 (EK1122)/IM2L0 AT2L0 SL1L0 JUNCTION (CU1124)/X2 AT2L0-SOLID (EK1100)/AT2L0-EL7041-04
//     PlcTask Inputs/Main.M4.bLimitBackwardEnable <-> STM Status/Status/Digital input 1
//     PlcTask Inputs/Main.M4.bLimitForwardEnable <-> STM Status/Status/Digital input 2
//   lfe_motion Instance <-> PLC Rail (EtherCAT)/Power (EK1200)/PLC Junction 2 (EK1122)/IM2L0 AT2L0 SL1L0 JUNCTION (CU1124)/X2 AT2L0-SOLID (EK1100)/AT2L0-EL7041-05
//     PlcTask Inputs/Main.M5.bLimitBackwardEnable <-> STM Status/Status/Digital input 1
//     PlcTask Inputs/Main.M5.bLimitForwardEnable <-> STM Status/Status/Digital input 2
//   lfe_motion Instance <-> PLC Rail (EtherCAT)/Power (EK1200)/PLC Junction 2 (EK1122)/IM2L0 AT2L0 SL1L0 JUNCTION (CU1124)/X2 AT2L0-SOLID (EK1100)/AT2L0-EL7041-06
//     PlcTask Inputs/Main.M6.bLimitBackwardEnable <-> STM Status/Status/Digital input 1
//     PlcTask Inputs/Main.M6.bLimitForwardEnable <-> STM Status/Status/Digital input 2
//   lfe_motion Instance <-> PLC Rail (EtherCAT)/Power (EK1200)/PLC Junction 2 (EK1122)/IM2L0 AT2L0 SL1L0 JUNCTION (CU1124)/X2 AT2L0-SOLID (EK1100)/AT2L0-EL7041-07
//     PlcTask Inputs/Main.M7.bLimitBackwardEnable <-> STM Status/Status/Digital input 1
//     PlcTask Inputs/Main.M7.bLimitForwardEnable <-> STM Status/Status/Digital input 2
//   lfe_motion Instance <-> PLC Rail (EtherCAT)/Power (EK1200)/PLC Junction 2 (EK1122)/IM2L0 AT2L0 SL1L0 JUNCTION (CU1124)/X2 AT2L0-SOLID (EK1100)/AT2L0-EL7041-08
//     PlcTask Inputs/Main.M8.bLimitBackwardEnable <-> STM Status/Status/Digital input 1
//     PlcTask Inputs/Main.M8.bLimitForwardEnable <-> STM Status/Status/Digital input 2
//   lfe_motion Instance <-> PLC Rail (EtherCAT)/Power (EK1200)/PLC Junction 2 (EK1122)/IM2L0 AT2L0 SL1L0 JUNCTION (CU1124)/X2 AT2L0-SOLID (EK1100)/AT2L0-EL7041-09
//     PlcTask Inputs/Main.M9.bLimitBackwardEnable <-> STM Status/Status/Digital input 1
//     PlcTask Inputs/Main.M9.bLimitForwardEnable <-> STM Status/Status/Digital input 2
//   lfe_motion Instance <-> PLC Rail (EtherCAT)/Power (EK1200)/PLC Junction 2 (EK1122)/IM2L0 AT2L0 SL1L0 JUNCTION (CU1124)/X2 AT2L0-SOLID (EK1100)/AT2L0-EL7041-10
//     PlcTask Inputs/Main.M10.bLimitBackwardEnable <-> STM Status/Status/Digital input 1
//     PlcTask Inputs/Main.M10.bLimitForwardEnable <-> STM Status/Status/Digital input 2
//   lfe_motion Instance <-> PLC Rail (EtherCAT)/Power (EK1200)/PLC Junction 2 (EK1122)/IM2L0 AT2L0 SL1L0 JUNCTION (CU1124)/X2 AT2L0-SOLID (EK1100)/AT2L0-EL7041-11
//     PlcTask Inputs/Main.M11.bLimitBackwardEnable <-> STM Status/Status/Digital input 1
//     PlcTask Inputs/Main.M11.bLimitForwardEnable <-> STM Status/Status/Digital input 2
//   lfe_motion Instance <-> PLC Rail (EtherCAT)/Power (EK1200)/PLC Junction 2 (EK1122)/IM2L0 AT2L0 SL1L0 JUNCTION (CU1124)/X2 AT2L0-SOLID (EK1100)/AT2L0-EL7041-12
//     PlcTask Inputs/Main.M12.bLimitBackwardEnable <-> STM Status/Status/Digital input 1
//     PlcTask Inputs/Main.M12.bLimitForwardEnable <-> STM Status/Status/Digital input 2
//   lfe_motion Instance <-> PLC Rail (EtherCAT)/Power (EK1200)/PLC Junction 2 (EK1122)/IM2L0 AT2L0 SL1L0 JUNCTION (CU1124)/X2 AT2L0-SOLID (EK1100)/AT2L0-EL7041-13
//     PlcTask Inputs/Main.M13.bLimitBackwardEnable <-> STM Status/Status/Digital input 1
//     PlcTask Inputs/Main.M13.bLimitForwardEnable <-> STM Status/Status/Digital input 2
//   lfe_motion Instance <-> PLC Rail (EtherCAT)/Power (EK1200)/PLC Junction 2 (EK1122)/IM2L0 AT2L0 SL1L0 JUNCTION (CU1124)/X2 AT2L0-SOLID (EK1100)/AT2L0-EL7041-14
//     PlcTask Inputs/Main.M14.bLimitBackwardEnable <-> STM Status/Status/Digital input 1
//     PlcTask Inputs/Main.M14.bLimitForwardEnable <-> STM Status/Status/Digital input 2
//   lfe_motion Instance <-> PLC Rail (EtherCAT)/Power (EK1200)/PLC Junction 2 (EK1122)/IM2L0 AT2L0 SL1L0 JUNCTION (CU1124)/X2 AT2L0-SOLID (EK1100)/AT2L0-EL7041-15
//     PlcTask Inputs/Main.M15.bLimitBackwardEnable <-> STM Status/Status/Digital input 1
//     PlcTask Inputs/Main.M15.bLimitForwardEnable <-> STM Status/Status/Digital input 2
//   lfe_motion Instance <-> PLC Rail (EtherCAT)/Power (EK1200)/PLC Junction 2 (EK1122)/IM2L0 AT2L0 SL1L0 JUNCTION (CU1124)/X2 AT2L0-SOLID (EK1100)/AT2L0-EL7041-16
//     PlcTask Inputs/Main.M16.bLimitBackwardEnable <-> STM Status/Status/Digital input 1
//     PlcTask Inputs/Main.M16.bLimitForwardEnable <-> STM Status/Status/Digital input 2
//   lfe_motion Instance <-> PLC Rail (EtherCAT)/Power (EK1200)/PLC Junction 2 (EK1122)/IM2L0 AT2L0 SL1L0 JUNCTION (CU1124)/X2 AT2L0-SOLID (EK1100)/AT2L0-EL7041-17
//     PlcTask Inputs/Main.M17.bLimitBackwardEnable <-> STM Status/Status/Digital input 1
//     PlcTask Inputs/Main.M17.bLimitForwardEnable <-> STM Status/Status/Digital input 2
//   lfe_motion Instance <-> PLC Rail (EtherCAT)/Power (EK1200)/PLC Junction 2 (EK1122)/IM2L0 AT2L0 SL1L0 JUNCTION (CU1124)/X2 AT2L0-SOLID (EK1100)/AT2L0-EL7041-18
//     PlcTask Inputs/Main.M18.bLimitBackwardEnable <-> STM Status/Status/Digital input 1
//     PlcTask Inputs/Main.M18.bLimitForwardEnable <-> STM Status/Status/Digital input 2
//   lfe_motion Instance <-> PLC Rail (EtherCAT)/Power (EK1200)/PLC Junction 2 (EK1122)/IM2L0 AT2L0 SL1L0 JUNCTION (CU1124)/X2 AT2L0-SOLID (EK1100)/AT2L0-EL7041-19
//     PlcTask Inputs/Main.M19.bLimitBackwardEnable <-> STM Status/Status/Digital input 1
//     PlcTask Inputs/Main.M19.bLimitForwardEnable <-> STM Status/Status/Digital input 2
//   lfe_motion Instance <-> PLC Rail (EtherCAT)/Power (EK1200)/PLC Junction 2 (EK1122)/X2 HXR EC2 (EK1100)/EC2 E1 (EK1122)/X1 IM3L0-PPM (EK1100)/IM3L0-EL2004
//     PlcTask Outputs/Main.M27.bBrakeRelease <-> Channel 1/Output
//     PlcTask Outputs/PRG_IM3L0_PPM.fbIM3L0.fbGige.bGigePower <-> Channel 2/Output
//   lfe_motion Instance <-> PLC Rail (EtherCAT)/Power (EK1200)/PLC Junction 2 (EK1122)/X2 HXR EC2 (EK1100)/EC2 E1 (EK1122)/X1 IM3L0-PPM (EK1100)/IM3L0-EL3062
//     PlcTask Inputs/PRG_IM3L0_PPM.fbIM3L0.fbPowerMeter.iVoltageINT <-> AI Standard Channel 1/Value
//   lfe_motion Instance <-> PLC Rail (EtherCAT)/Power (EK1200)/PLC Junction 2 (EK1122)/X2 HXR EC2 (EK1100)/EC2 E1 (EK1122)/X1 IM3L0-PPM (EK1100)/IM3L0-EL3314
//     PlcTask Inputs/PRG_IM3L0_PPM.fbIM3L0.fbPowerMeter.fbTempSensor.bError <-> TC Inputs Channel 1/Status/Error
//     PlcTask Inputs/PRG_IM3L0_PPM.fbIM3L0.fbPowerMeter.fbTempSensor.bOverrange <-> TC Inputs Channel 1/Status/Overrange
//     PlcTask Inputs/PRG_IM3L0_PPM.fbIM3L0.fbPowerMeter.fbTempSensor.bUnderrange <-> TC Inputs Channel 1/Status/Underrange
//     PlcTask Inputs/PRG_IM3L0_PPM.fbIM3L0.fbPowerMeter.fbTempSensor.iRaw <-> TC Inputs Channel 1/Value
//     PlcTask Inputs/PRG_IM3L0_PPM.fbIM3L0.fbYagTempSensor.bError <-> TC Inputs Channel 2/Status/Error
//     PlcTask Inputs/PRG_IM3L0_PPM.fbIM3L0.fbYagTempSensor.bOverrange <-> TC Inputs Channel 2/Status/Overrange
//     PlcTask Inputs/PRG_IM3L0_PPM.fbIM3L0.fbYagTempSensor.bUnderrange <-> TC Inputs Channel 2/Status/Underrange
//     PlcTask Inputs/PRG_IM3L0_PPM.fbIM3L0.fbYagTempSensor.iRaw <-> TC Inputs Channel 2/Value
//   lfe_motion Instance <-> PLC Rail (EtherCAT)/Power (EK1200)/PLC Junction 2 (EK1122)/X2 HXR EC2 (EK1100)/EC2 E1 (EK1122)/X1 IM3L0-PPM (EK1100)/IM3L0-EL4004
//     PlcTask Outputs/PRG_IM3L0_PPM.fbIM3L0.fbGige.iIlluminatorINT <-> AO Outputs Channel 1/Analog output
//   lfe_motion Instance <-> PLC Rail (EtherCAT)/Power (EK1200)/PLC Junction 2 (EK1122)/X2 HXR EC2 (EK1100)/EC2 E1 (EK1122)/X1 IM3L0-PPM (EK1100)/IM3L0-EL7041
//     PlcTask Inputs/Main.M27.bLimitBackwardEnable <-> STM Status/Status/Digital input 2
//     PlcTask Inputs/Main.M27.bLimitForwardEnable <-> STM Status/Status/Digital input 1
//   lfe_motion Instance <-> PLC Rail (EtherCAT)/Power (EK1200)/PLC Junction 2 (EK1122)/X2 HXR EC2 (EK1100)/EC2 E1 (EK1122)/X2 IM1L1-PPM (EK1100)/IM1L1-EL2004
//     PlcTask Outputs/Main.M23.bBrakeRelease <-> Channel 1/Output
//     PlcTask Outputs/PRG_IM1L1_PPM.fbIM1L1.fbGige.bGigePower <-> Channel 2/Output
//   lfe_motion Instance <-> PLC Rail (EtherCAT)/Power (EK1200)/PLC Junction 2 (EK1122)/X2 HXR EC2 (EK1100)/EC2 E1 (EK1122)/X2 IM1L1-PPM (EK1100)/IM1L1-EL3062
//     PlcTask Inputs/PRG_IM1L1_PPM.fbIM1L1.fbPowerMeter.iVoltageINT <-> AI Standard Channel 1/Value
//   lfe_motion Instance <-> PLC Rail (EtherCAT)/Power (EK1200)/PLC Junction 2 (EK1122)/X2 HXR EC2 (EK1100)/EC2 E1 (EK1122)/X2 IM1L1-PPM (EK1100)/IM1L1-EL3314
//     PlcTask Inputs/PRG_IM1L1_PPM.fbIM1L1.fbPowerMeter.fbTempSensor.bError <-> TC Inputs Channel 1/Status/Error
//     PlcTask Inputs/PRG_IM1L1_PPM.fbIM1L1.fbPowerMeter.fbTempSensor.bOverrange <-> TC Inputs Channel 1/Status/Overrange
//     PlcTask Inputs/PRG_IM1L1_PPM.fbIM1L1.fbPowerMeter.fbTempSensor.bUnderrange <-> TC Inputs Channel 1/Status/Underrange
//     PlcTask Inputs/PRG_IM1L1_PPM.fbIM1L1.fbPowerMeter.fbTempSensor.iRaw <-> TC Inputs Channel 1/Value
//     PlcTask Inputs/PRG_IM1L1_PPM.fbIM1L1.fbYagTempSensor.bError <-> TC Inputs Channel 2/Status/Error
//     PlcTask Inputs/PRG_IM1L1_PPM.fbIM1L1.fbYagTempSensor.bOverrange <-> TC Inputs Channel 2/Status/Overrange
//     PlcTask Inputs/PRG_IM1L1_PPM.fbIM1L1.fbYagTempSensor.bUnderrange <-> TC Inputs Channel 2/Status/Underrange
//     PlcTask Inputs/PRG_IM1L1_PPM.fbIM1L1.fbYagTempSensor.iRaw <-> TC Inputs Channel 2/Value
//   lfe_motion Instance <-> PLC Rail (EtherCAT)/Power (EK1200)/PLC Junction 2 (EK1122)/X2 HXR EC2 (EK1100)/EC2 E1 (EK1122)/X2 IM1L1-PPM (EK1100)/IM1L1-EL4004
//     PlcTask Outputs/PRG_IM1L1_PPM.fbIM1L1.fbGige.iIlluminatorINT <-> AO Outputs Channel 1/Analog output
//   lfe_motion Instance <-> PLC Rail (EtherCAT)/Power (EK1200)/PLC Junction 2 (EK1122)/X2 HXR EC2 (EK1100)/EC2 E1 (EK1122)/X2 IM1L1-PPM (EK1100)/IM1L1-EL7041
//     PlcTask Inputs/Main.M23.bLimitBackwardEnable <-> STM Status/Status/Digital input 2
//     PlcTask Inputs/Main.M23.bLimitForwardEnable <-> STM Status/Status/Digital input 1
//   lfe_motion Instance <-> PLC Rail (EtherCAT)/Power (EK1200)/PLC Junction 2 (EK1122)/X2 HXR EC2 (EK1100)/EC2 E2 (EK1122)/X1 IM4L0-XTES (EK1100)/IM4L0-EL1088
//     PlcTask Inputs/Main.M29.bHome <-> Channel 2/Input
//     PlcTask Inputs/Main.M30.bHome <-> Channel 4/Input
//     PlcTask Inputs/PRG_IM4L0_XTES.fbIM4L0.bFocusEndBwd <-> Channel 4/Input
//     PlcTask Inputs/PRG_IM4L0_XTES.fbIM4L0.bFocusEndFwd <-> Channel 3/Input
//     PlcTask Inputs/PRG_IM4L0_XTES.fbIM4L0.bZoomEndBwd <-> Channel 2/Input
//     PlcTask Inputs/PRG_IM4L0_XTES.fbIM4L0.bZoomEndFwd <-> Channel 1/Input
//   lfe_motion Instance <-> PLC Rail (EtherCAT)/Power (EK1200)/PLC Junction 2 (EK1122)/X2 HXR EC2 (EK1100)/EC2 E2 (EK1122)/X1 IM4L0-XTES (EK1100)/IM4L0-EL2004
//     PlcTask Outputs/Main.M28.bBrakeRelease <-> Channel 1/Output
//     PlcTask Outputs/PRG_IM4L0_XTES.bIM4L0_SCRP_LED_01 <-> Channel 4/Output
//     PlcTask Outputs/PRG_IM4L0_XTES.fbIM4L0.fbLED.bLEDPower <-> Channel 3/Output
//     PlcTask Outputs/PRG_IM4L0_XTES.fbIM4L0.fbOpal.bOpalPower <-> Channel 2/Output
//   lfe_motion Instance <-> PLC Rail (EtherCAT)/Power (EK1200)/PLC Junction 2 (EK1122)/X2 HXR EC2 (EK1100)/EC2 E2 (EK1122)/X1 IM4L0-XTES (EK1100)/IM4L0-EL6002
//     PlcTask Inputs/PRG_IM4L0_XTES.stEL6In/D[{0..21}] <-> COM TxPDO-Map Inputs Channel 1/Data In {0..21}  (22 links)
//     PlcTask Inputs/PRG_IM4L0_XTES.stEL6In/Status <-> COM TxPDO-Map Inputs Channel 1/Status
//     PlcTask Outputs/PRG_IM4L0_XTES.stEL6Out/Ctrl <-> COM RxPDO-Map Outputs Channel 1/Ctrl
//     PlcTask Outputs/PRG_IM4L0_XTES.stEL6Out/D[{0..21}] <-> COM RxPDO-Map Outputs Channel 1/Data Out {0..21}  (22 links)
//   lfe_motion Instance <-> PLC Rail (EtherCAT)/Power (EK1200)/PLC Junction 2 (EK1122)/X2 HXR EC2 (EK1100)/EC2 E2 (EK1122)/X1 IM4L0-XTES (EK1100)/IM4L0-EL7041
//     PlcTask Inputs/Main.M28.bLimitForwardEnable <-> STM Status/Status/Digital input 1
//   lfe_motion Instance <-> PLC Rail (EtherCAT)/Power (EK1200)/PLC Junction 2 (EK1122)/X2 HXR EC2 (EK1100)/EC2 E2 (EK1122)/X2 ECJ (CU1128)/X2 EM3L0-IPM (EK1100)/EM3L0-EL2004-E4
//     PlcTask Outputs/Main.M56.bBrakeRelease <-> Channel 1/Output
//   lfe_motion Instance <-> PLC Rail (EtherCAT)/Power (EK1200)/PLC Junction 2 (EK1122)/X2 HXR EC2 (EK1100)/EC2 E2 (EK1122)/X2 ECJ (CU1128)/X2 EM3L0-IPM (EK1100)/EM3L0-EL5042-E2
//     PlcTask Inputs/Main.M55.nRawEncoderULINT <-> FB Inputs Channel 1/Position
//     PlcTask Inputs/Main.M56.nRawEncoderULINT <-> FB Inputs Channel 2/Position
//   lfe_motion Instance <-> PLC Rail (EtherCAT)/Power (EK1200)/PLC Junction 2 (EK1122)/X2 SL2L0-Power (EK1100)/SL2L0-EL3202-E10
//     PlcTask Inputs/PRG_SL2L0_POWER.fbSL2L0.RTD_North_1.bError <-> RTD Inputs Channel 1/Status/Error
//     PlcTask Inputs/PRG_SL2L0_POWER.fbSL2L0.RTD_North_1.iRaw <-> RTD Inputs Channel 1/Value
//     PlcTask Inputs/PRG_SL2L0_POWER.fbSL2L0.RTD_TOP_1.bError <-> RTD Inputs Channel 1/Status/Error
//     PlcTask Inputs/PRG_SL2L0_POWER.fbSL2L0.RTD_TOP_2.bError <-> RTD Inputs Channel 2/Status/Error
//     PlcTask Inputs/PRG_SL2L0_POWER.fbSL2L0.RTD_TOP_1.bOverrange <-> RTD Inputs Channel 1/Status/Overrange
//     PlcTask Inputs/PRG_SL2L0_POWER.fbSL2L0.RTD_TOP_2.bOverrange <-> RTD Inputs Channel 2/Status/Overrange
//     PlcTask Inputs/PRG_SL2L0_POWER.fbSL2L0.RTD_TOP_1.bUnderrange <-> RTD Inputs Channel 1/Status/Underrange
//     PlcTask Inputs/PRG_SL2L0_POWER.fbSL2L0.RTD_TOP_2.bUnderrange <-> RTD Inputs Channel 2/Status/Underrange
//     PlcTask Inputs/PRG_SL2L0_POWER.fbSL2L0.RTD_TOP_1.iRaw <-> RTD Inputs Channel 1/Value
//     PlcTask Inputs/PRG_SL2L0_POWER.fbSL2L0.RTD_TOP_2.iRaw <-> RTD Inputs Channel 2/Value
//   lfe_motion Instance <-> PLC Rail (EtherCAT)/Power (EK1200)/PLC Junction 2 (EK1122)/X2 SL2L0-Power (EK1100)/SL2L0-EL3202-E11
//     PlcTask Inputs/PRG_SL2L0_POWER.fbSL2L0.RTD_North_1.bOverrange <-> RTD Inputs Channel 1/Status/Overrange
//     PlcTask Inputs/PRG_SL2L0_POWER.fbSL2L0.RTD_North_2.bOverrange <-> RTD Inputs Channel 2/Status/Overrange
//     PlcTask Inputs/PRG_SL2L0_POWER.fbSL2L0.RTD_North_1.bUnderrange <-> RTD Inputs Channel 1/Status/Underrange
//     PlcTask Inputs/PRG_SL2L0_POWER.fbSL2L0.RTD_North_2.bUnderrange <-> RTD Inputs Channel 2/Status/Underrange
//     PlcTask Inputs/PRG_SL2L0_POWER.fbSL2L0.RTD_North_2.bError <-> RTD Inputs Channel 2/Status/Error
//     PlcTask Inputs/PRG_SL2L0_POWER.fbSL2L0.RTD_North_2.iRaw <-> RTD Inputs Channel 2/Value
//   lfe_motion Instance <-> PLC Rail (EtherCAT)/Power (EK1200)/PLC Junction 2 (EK1122)/X2 SL2L0-Power (EK1100)/SL2L0-EL3202-E8
//     PlcTask Inputs/PRG_SL2L0_POWER.fbSL2L0.RTD_Bottom_1.bError <-> RTD Inputs Channel 1/Status/Error
//     PlcTask Inputs/PRG_SL2L0_POWER.fbSL2L0.RTD_Bottom_2.bError <-> RTD Inputs Channel 2/Status/Error
//     PlcTask Inputs/PRG_SL2L0_POWER.fbSL2L0.RTD_Bottom_1.bOverrange <-> RTD Inputs Channel 1/Status/Overrange
//     PlcTask Inputs/PRG_SL2L0_POWER.fbSL2L0.RTD_Bottom_2.bOverrange <-> RTD Inputs Channel 2/Status/Overrange
//     PlcTask Inputs/PRG_SL2L0_POWER.fbSL2L0.RTD_Bottom_1.bUnderrange <-> RTD Inputs Channel 1/Status/Underrange
//     PlcTask Inputs/PRG_SL2L0_POWER.fbSL2L0.RTD_Bottom_2.bUnderrange <-> RTD Inputs Channel 2/Status/Underrange
//     PlcTask Inputs/PRG_SL2L0_POWER.fbSL2L0.RTD_Bottom_1.iRaw <-> RTD Inputs Channel 1/Value
//     PlcTask Inputs/PRG_SL2L0_POWER.fbSL2L0.RTD_Bottom_2.iRaw <-> RTD Inputs Channel 2/Value
//   lfe_motion Instance <-> PLC Rail (EtherCAT)/Power (EK1200)/PLC Junction 2 (EK1122)/X2 SL2L0-Power (EK1100)/SL2L0-EL3202-E9
//     PlcTask Inputs/PRG_SL2L0_POWER.fbSL2L0.RTD_South_1.bError <-> RTD Inputs Channel 1/Status/Error
//     PlcTask Inputs/PRG_SL2L0_POWER.fbSL2L0.RTD_South_2.bError <-> RTD Inputs Channel 2/Status/Error
//     PlcTask Inputs/PRG_SL2L0_POWER.fbSL2L0.RTD_South_1.bOverrange <-> RTD Inputs Channel 1/Status/Overrange
//     PlcTask Inputs/PRG_SL2L0_POWER.fbSL2L0.RTD_South_2.bOverrange <-> RTD Inputs Channel 2/Status/Overrange
//     PlcTask Inputs/PRG_SL2L0_POWER.fbSL2L0.RTD_South_1.bUnderrange <-> RTD Inputs Channel 1/Status/Underrange
//     PlcTask Inputs/PRG_SL2L0_POWER.fbSL2L0.RTD_South_2.bUnderrange <-> RTD Inputs Channel 2/Status/Underrange
//     PlcTask Inputs/PRG_SL2L0_POWER.fbSL2L0.RTD_South_1.iRaw <-> RTD Inputs Channel 1/Value
//     PlcTask Inputs/PRG_SL2L0_POWER.fbSL2L0.RTD_South_2.iRaw <-> RTD Inputs Channel 2/Value
//   lfe_motion Instance <-> PLC Rail (EtherCAT)/Power (EK1200)/PLC Junction 2 (EK1122)/X2 SL2L0-Power (EK1100)/SL2L0-EL7041-E1
//     PlcTask Inputs/Main.M45.bLimitBackwardEnable <-> STM Status/Status/Digital input 1
//     PlcTask Inputs/Main.M45.bLimitForwardEnable <-> STM Status/Status/Digital input 2
//   lfe_motion Instance <-> PLC Rail (EtherCAT)/Power (EK1200)/PLC Junction 2 (EK1122)/X2 SL2L0-Power (EK1100)/SL2L0-EL7041-E3
//     PlcTask Inputs/Main.M46.bLimitBackwardEnable <-> STM Status/Status/Digital input 2
//     PlcTask Inputs/Main.M46.bLimitForwardEnable <-> STM Status/Status/Digital input 1
//   lfe_motion Instance <-> PLC Rail (EtherCAT)/Power (EK1200)/PLC Junction 2 (EK1122)/X2 SL2L0-Power (EK1100)/SL2L0-EL7041-E5
//     PlcTask Inputs/Main.M47.bLimitBackwardEnable <-> STM Status/Status/Digital input 1
//     PlcTask Inputs/Main.M47.bLimitForwardEnable <-> STM Status/Status/Digital input 2
//   lfe_motion Instance <-> PLC Rail (EtherCAT)/Power (EK1200)/PLC Junction 2 (EK1122)/X2 SL2L0-Power (EK1100)/SL2L0-EL7041-E7
//     PlcTask Inputs/Main.M48.bLimitBackwardEnable <-> STM Status/Status/Digital input 2
//     PlcTask Inputs/Main.M48.bLimitForwardEnable <-> STM Status/Status/Digital input 1
//   lfe_motion Instance <-> PLC Rail (EtherCAT)/Power (EK1200)/PLC Junction 3  (EK1122)/X1 B950-100H2-L0S5-ECJ-01/B950-100H2-L0S5-ECJ-01 (CU1128-B)/AL1L0-REF/AL1L0-EL4004-E4
//     PlcTask Outputs/PRG_AL1L0_REF.fbAL1L0.fbLaser.iLaserINT <-> AO Outputs Channel 1/Analog output
//     PlcTask Outputs/PRG_AL1L0_REF.fbAL1L0.fbLaser.iShutdownINT <-> AO Outputs Channel 2/Analog output
//   lfe_motion Instance <-> PLC Rail (EtherCAT)/Power (EK1200)/PLC Junction 3  (EK1122)/X1 B950-100H2-L0S5-ECJ-01/B950-100H2-L0S5-ECJ-01 (CU1128-B)/AL1L0-REF/AL1L0-EL5042-E2
//     PlcTask Inputs/Main.M58.nRawEncoderULINT <-> FB Inputs Channel 2/Position
//   lfe_motion Instance <-> PLC Rail (EtherCAT)/Power (EK1200)/PLC Junction 3  (EK1122)/X1 B950-100H2-L0S5-ECJ-01/IM5L0-PPM/IM5L0-EL1084-E4
//     PlcTask Inputs/Main.M57.bLimitBackwardEnable <-> Channel 4/Input
//     PlcTask Inputs/Main.M57.bLimitForwardEnable <-> Channel 3/Input
//   lfe_motion Instance <-> PLC Rail (EtherCAT)/Power (EK1200)/PLC Junction 3  (EK1122)/X1 B950-100H2-L0S5-ECJ-01/IM5L0-PPM/IM5L0-EL2004-E3
//     PlcTask Outputs/Main.M57.bBrakeRelease <-> Channel 1/Output
//   lfe_motion Instance <-> PLC Rail (EtherCAT)/Power (EK1200)/PLC Junction 3  (EK1122)/X1 B950-100H2-L0S5-ECJ-01/IM5L0-PPM/IM5L0-EL3202-0010-E5
//     PlcTask Inputs/PRG_IM5L0_PPM.fbIM5L0.fbPowerMeter.fbTempSensor.bError <-> RTD Inputs Channel 1/Status/Error
//     PlcTask Inputs/PRG_IM5L0_PPM.fbIM5L0.fbPowerMeter.fbTempSensor.bOverrange <-> RTD Inputs Channel 1/Status/Overrange
//     PlcTask Inputs/PRG_IM5L0_PPM.fbIM5L0.fbPowerMeter.fbTempSensor.bUnderrange <-> RTD Inputs Channel 1/Status/Underrange
//     PlcTask Inputs/PRG_IM5L0_PPM.fbIM5L0.fbPowerMeter.fbTempSensor.iRaw <-> RTD Inputs Channel 1/Value
//   lfe_motion Instance <-> PLC Rail (EtherCAT)/Power (EK1200)/PLC Junction 3  (EK1122)/X1 B950-100H2-L0S5-ECJ-01/IM5L0-PPM/IM5L0-EL3602-E6
//     PlcTask Inputs/PRG_IM5L0_PPM.fbIM5L0.fbPowerMeter.iVoltageINT <-> AI Inputs Channel 1/Value
//   lfe_motion Instance <-> PLC Rail (EtherCAT)/Power (EK1200)/PLC Junction 3  (EK1122)/X1 B950-100H2-L0S5-ECJ-01/IM5L0-PPM/IM5L0-EL4004-E7
//     PlcTask Outputs/PRG_IM5L0_PPM.fbIM5L0.fbGige.iIlluminatorINT <-> AO Outputs Channel 1/Analog output
//   lfe_motion Instance <-> PLC Rail (EtherCAT)/Power (EK1200)/PLC Junction 3  (EK1122)/X1 B950-100H2-L0S5-ECJ-01/IM5L0-PPM/IM5L0-EL5042-E2
//     PlcTask Inputs/Main.M57.nRawEncoderULINT <-> FB Inputs Channel 1/Position
//   lfe_motion Instance <-> PLC Rail (EtherCAT)/Power (EK1200)/PLC Junction 3  (EK1122)/X1 B950-100H2-L0S5-ECJ-01/SL3L0-SCATTER/SL3L0-EL5042-E2
//     PlcTask Inputs/Main.M61.nRawEncoderULINT <-> FB Inputs Channel 1/Position
//     PlcTask Inputs/Main.M62.nRawEncoderULINT <-> FB Inputs Channel 2/Position
//   lfe_motion Instance <-> PLC Rail (EtherCAT)/Power (EK1200)/PLC Junction 3  (EK1122)/X1 B950-100H2-L0S5-ECJ-01/SL3L0-SCATTER/SL3L0-EL5042-E5
//     PlcTask Inputs/Main.M59.nRawEncoderULINT <-> FB Inputs Channel 1/Position
//     PlcTask Inputs/Main.M60.nRawEncoderULINT <-> FB Inputs Channel 2/Position
//   lfe_motion Instance <-> PLC Rail (EtherCAT)/Power (EK1200)/PLC Junction 3  (EK1122)/X1 B950-100H2-L0S5-ECJ-01/SL3L0-SCATTER/SL3L0-EL7037-E1
//     PlcTask Inputs/Main.M62.bLimitBackwardEnable <-> STM Status/Status/Digital input 2
//     PlcTask Inputs/Main.M62.bLimitForwardEnable <-> STM Status/Status/Digital input 1
//   lfe_motion Instance <-> PLC Rail (EtherCAT)/Power (EK1200)/PLC Junction 3  (EK1122)/X1 B950-100H2-L0S5-ECJ-01/SL3L0-SCATTER/SL3L0-EL7037-E3
//     PlcTask Inputs/Main.M61.bLimitBackwardEnable <-> STM Status/Status/Digital input 2
//     PlcTask Inputs/Main.M61.bLimitForwardEnable <-> STM Status/Status/Digital input 1
//   lfe_motion Instance <-> PLC Rail (EtherCAT)/Power (EK1200)/PLC Junction 3  (EK1122)/X1 B950-100H2-L0S5-ECJ-01/SL3L0-SCATTER/SL3L0-EL7037-E4
//     PlcTask Inputs/Main.M60.bLimitBackwardEnable <-> STM Status/Status/Digital input 2
//     PlcTask Inputs/Main.M60.bLimitForwardEnable <-> STM Status/Status/Digital input 1
//   lfe_motion Instance <-> PLC Rail (EtherCAT)/Power (EK1200)/PLC Junction 3  (EK1122)/X1 B950-100H2-L0S5-ECJ-01/SL3L0-SCATTER/SL3L0-EL7037-E6
//     PlcTask Inputs/Main.M59.bLimitBackwardEnable <-> STM Status/Status/Digital input 2
//     PlcTask Inputs/Main.M59.bLimitForwardEnable <-> STM Status/Status/Digital input 1
//   lfe_motion Instance <-> PLC Rail (EtherCAT)/Power (EK1200)/PMPS_FFO
//     PlcTask Outputs/GVL.fbFastFaultOutput1.q_xFastFaultOut <-> Channel 1/Output
//     PlcTask Outputs/GVL.fbFastFaultOutput2.q_xFastFaultOut <-> Channel 2/Output
//   lfe_motion Instance <-> PLC Rail (EtherCAT)/Power (EK1200)/PMPS_PRE
//     PlcTask Inputs/GVL.rReqTrans <-> IO Inputs/SattArrayReq
//     PlcTask Inputs/PRG_3_PMPS_POST.fbArbiterIO.i_stCurrentBP <-> IO Inputs/CurrentBP
//     PlcTask Inputs/PRG_3_PMPS_POST.fbArbiterIO.xTxPDO_state <-> SYNC Inputs/TxPDO state
//     PlcTask Inputs/PRG_3_PMPS_POST.fbArbiterIO.xTxPDO_toggle <-> SYNC Inputs/TxPDO toggle
//     PlcTask Outputs/GVL.rCurTrans <-> IO Outputs/SattArrayStatus
//     PlcTask Outputs/PRG_3_PMPS_POST.fbArbiterIO.q_stRequestedBP <-> IO Outputs/RequestedBP
//   lfe_motion Instance <-> NC-Task 1 SAF/Axes/AL1L0-REF-MMS-M58
//     PlcTask Inputs/Main.M58.Axis.NcToPlc <-> Outputs/ToPlc
//     PlcTask Outputs/Main.M58.Axis.PlcToNc <-> Inputs/FromPlc
//   lfe_motion Instance <-> NC-Task 1 SAF/Axes/Axis 1
//     PlcTask Inputs/Main.M1.Axis.NcToPlc <-> Outputs/ToPlc
//     PlcTask Outputs/Main.M1.Axis.PlcToNc <-> Inputs/FromPlc
//   lfe_motion Instance <-> NC-Task 1 SAF/Axes/Axis 10
//     PlcTask Inputs/Main.M10.Axis.NcToPlc <-> Outputs/ToPlc
//     PlcTask Outputs/Main.M10.Axis.PlcToNc <-> Inputs/FromPlc
//   lfe_motion Instance <-> NC-Task 1 SAF/Axes/Axis 11
//     PlcTask Inputs/Main.M11.Axis.NcToPlc <-> Outputs/ToPlc
//     PlcTask Outputs/Main.M11.Axis.PlcToNc <-> Inputs/FromPlc
//   lfe_motion Instance <-> NC-Task 1 SAF/Axes/Axis 12
//     PlcTask Inputs/Main.M12.Axis.NcToPlc <-> Outputs/ToPlc
//     PlcTask Outputs/Main.M12.Axis.PlcToNc <-> Inputs/FromPlc
//   lfe_motion Instance <-> NC-Task 1 SAF/Axes/Axis 13
//     PlcTask Inputs/Main.M13.Axis.NcToPlc <-> Outputs/ToPlc
//     PlcTask Outputs/Main.M13.Axis.PlcToNc <-> Inputs/FromPlc
//   lfe_motion Instance <-> NC-Task 1 SAF/Axes/Axis 14
//     PlcTask Inputs/Main.M14.Axis.NcToPlc <-> Outputs/ToPlc
//     PlcTask Outputs/Main.M14.Axis.PlcToNc <-> Inputs/FromPlc
//   lfe_motion Instance <-> NC-Task 1 SAF/Axes/Axis 15
//     PlcTask Inputs/Main.M15.Axis.NcToPlc <-> Outputs/ToPlc
//     PlcTask Outputs/Main.M15.Axis.PlcToNc <-> Inputs/FromPlc
//   lfe_motion Instance <-> NC-Task 1 SAF/Axes/Axis 16
//     PlcTask Inputs/Main.M16.Axis.NcToPlc <-> Outputs/ToPlc
//     PlcTask Outputs/Main.M16.Axis.PlcToNc <-> Inputs/FromPlc
//   lfe_motion Instance <-> NC-Task 1 SAF/Axes/Axis 17
//     PlcTask Inputs/Main.M17.Axis.NcToPlc <-> Outputs/ToPlc
//     PlcTask Outputs/Main.M17.Axis.PlcToNc <-> Inputs/FromPlc
//   lfe_motion Instance <-> NC-Task 1 SAF/Axes/Axis 18
//     PlcTask Inputs/Main.M18.Axis.NcToPlc <-> Outputs/ToPlc
//     PlcTask Outputs/Main.M18.Axis.PlcToNc <-> Inputs/FromPlc
//   lfe_motion Instance <-> NC-Task 1 SAF/Axes/Axis 19
//     PlcTask Inputs/Main.M19.Axis.NcToPlc <-> Outputs/ToPlc
//     PlcTask Outputs/Main.M19.Axis.PlcToNc <-> Inputs/FromPlc
//   lfe_motion Instance <-> NC-Task 1 SAF/Axes/Axis 2
//     PlcTask Inputs/Main.M2.Axis.NcToPlc <-> Outputs/ToPlc
//     PlcTask Outputs/Main.M2.Axis.PlcToNc <-> Inputs/FromPlc
//   lfe_motion Instance <-> NC-Task 1 SAF/Axes/Axis 20 IM1L0-XTES-MMS
//     PlcTask Inputs/Main.M20.Axis.NcToPlc <-> Outputs/ToPlc
//     PlcTask Outputs/Main.M20.Axis.PlcToNc <-> Inputs/FromPlc
//   lfe_motion Instance <-> NC-Task 1 SAF/Axes/Axis 21 IM1L0-XTES-CLZ
//     PlcTask Inputs/Main.M21.Axis.NcToPlc <-> Outputs/ToPlc
//     PlcTask Outputs/Main.M21.Axis.PlcToNc <-> Inputs/FromPlc
//   lfe_motion Instance <-> NC-Task 1 SAF/Axes/Axis 22 IM1L0-XTES-CLF
//     PlcTask Inputs/Main.M22.Axis.NcToPlc <-> Outputs/ToPlc
//     PlcTask Outputs/Main.M22.Axis.PlcToNc <-> Inputs/FromPlc
//   lfe_motion Instance <-> NC-Task 1 SAF/Axes/Axis 23 IM1L1-PPM-MMS
//     PlcTask Inputs/Main.M23.Axis.NcToPlc <-> Outputs/ToPlc
//     PlcTask Outputs/Main.M23.Axis.PlcToNc <-> Inputs/FromPlc
//   lfe_motion Instance <-> NC-Task 1 SAF/Axes/Axis 24 IM2L0-XTES-MMS
//     PlcTask Inputs/Main.M24.Axis.NcToPlc <-> Outputs/ToPlc
//     PlcTask Outputs/Main.M24.Axis.PlcToNc <-> Inputs/FromPlc
//   lfe_motion Instance <-> NC-Task 1 SAF/Axes/Axis 25 IM2L0-XTES-CLZ
//     PlcTask Inputs/Main.M25.Axis.NcToPlc <-> Outputs/ToPlc
//     PlcTask Outputs/Main.M25.Axis.PlcToNc <-> Inputs/FromPlc
//   lfe_motion Instance <-> NC-Task 1 SAF/Axes/Axis 26 IM2L0-XTES-CLF
//     PlcTask Inputs/Main.M26.Axis.NcToPlc <-> Outputs/ToPlc
//     PlcTask Outputs/Main.M26.Axis.PlcToNc <-> Inputs/FromPlc
//   lfe_motion Instance <-> NC-Task 1 SAF/Axes/Axis 27 IM3L0-PPM-MMS
//     PlcTask Inputs/Main.M27.Axis.NcToPlc <-> Outputs/ToPlc
//     PlcTask Outputs/Main.M27.Axis.PlcToNc <-> Inputs/FromPlc
//   lfe_motion Instance <-> NC-Task 1 SAF/Axes/Axis 28 IM4L0-XTES-MMS
//     PlcTask Inputs/Main.M28.Axis.NcToPlc <-> Outputs/ToPlc
//     PlcTask Outputs/Main.M28.Axis.PlcToNc <-> Inputs/FromPlc
//   lfe_motion Instance <-> NC-Task 1 SAF/Axes/Axis 29 IM4L0-XTES-CLZ
//     PlcTask Inputs/Main.M29.Axis.NcToPlc <-> Outputs/ToPlc
//     PlcTask Outputs/Main.M29.Axis.PlcToNc <-> Inputs/FromPlc
//   lfe_motion Instance <-> NC-Task 1 SAF/Axes/Axis 3
//     PlcTask Inputs/Main.M3.Axis.NcToPlc <-> Outputs/ToPlc
//     PlcTask Outputs/Main.M3.Axis.PlcToNc <-> Inputs/FromPlc
//   lfe_motion Instance <-> NC-Task 1 SAF/Axes/Axis 30 IM4L0-XTES-CLF
//     PlcTask Inputs/Main.M30.Axis.NcToPlc <-> Outputs/ToPlc
//     PlcTask Outputs/Main.M30.Axis.PlcToNc <-> Inputs/FromPlc
//   lfe_motion Instance <-> NC-Task 1 SAF/Axes/Axis 33
//     PlcTask Inputs/Main.M33.Axis.NcToPlc <-> Outputs/ToPlc
//     PlcTask Outputs/Main.M33.Axis.PlcToNc <-> Inputs/FromPlc
//   lfe_motion Instance <-> NC-Task 1 SAF/Axes/Axis 34
//     PlcTask Inputs/Main.M34.Axis.NcToPlc <-> Outputs/ToPlc
//     PlcTask Outputs/Main.M34.Axis.PlcToNc <-> Inputs/FromPlc
//   lfe_motion Instance <-> NC-Task 1 SAF/Axes/Axis 35
//     PlcTask Inputs/Main.M35.Axis.NcToPlc <-> Outputs/ToPlc
//     PlcTask Outputs/Main.M35.Axis.PlcToNc <-> Inputs/FromPlc
//   lfe_motion Instance <-> NC-Task 1 SAF/Axes/Axis 36
//     PlcTask Inputs/Main.M36.Axis.NcToPlc <-> Outputs/ToPlc
//     PlcTask Outputs/Main.M36.Axis.PlcToNc <-> Inputs/FromPlc
//   lfe_motion Instance <-> NC-Task 1 SAF/Axes/Axis 37
//     PlcTask Inputs/Main.M37.Axis.NcToPlc <-> Outputs/ToPlc
//     PlcTask Outputs/Main.M37.Axis.PlcToNc <-> Inputs/FromPlc
//   lfe_motion Instance <-> NC-Task 1 SAF/Axes/Axis 38
//     PlcTask Inputs/Main.M38.Axis.NcToPlc <-> Outputs/ToPlc
//     PlcTask Outputs/Main.M38.Axis.PlcToNc <-> Inputs/FromPlc
//   lfe_motion Instance <-> NC-Task 1 SAF/Axes/Axis 39
//     PlcTask Inputs/Main.M39.Axis.NcToPlc <-> Outputs/ToPlc
//     PlcTask Outputs/Main.M39.Axis.PlcToNc <-> Inputs/FromPlc
//   lfe_motion Instance <-> NC-Task 1 SAF/Axes/Axis 4
//     PlcTask Inputs/Main.M4.Axis.NcToPlc <-> Outputs/ToPlc
//     PlcTask Outputs/Main.M4.Axis.PlcToNc <-> Inputs/FromPlc
//   lfe_motion Instance <-> NC-Task 1 SAF/Axes/Axis 40
//     PlcTask Inputs/Main.M40.Axis.NcToPlc <-> Outputs/ToPlc
//     PlcTask Outputs/Main.M40.Axis.PlcToNc <-> Inputs/FromPlc
//   lfe_motion Instance <-> NC-Task 1 SAF/Axes/Axis 5
//     PlcTask Inputs/Main.M5.Axis.NcToPlc <-> Outputs/ToPlc
//     PlcTask Outputs/Main.M5.Axis.PlcToNc <-> Inputs/FromPlc
//   lfe_motion Instance <-> NC-Task 1 SAF/Axes/Axis 57 IM5L0-PPM-MMS
//     PlcTask Inputs/Main.M57.Axis.NcToPlc <-> Outputs/ToPlc
//     PlcTask Outputs/Main.M57.Axis.PlcToNc <-> Inputs/FromPlc
//   lfe_motion Instance <-> NC-Task 1 SAF/Axes/Axis 6
//     PlcTask Inputs/Main.M6.Axis.NcToPlc <-> Outputs/ToPlc
//     PlcTask Outputs/Main.M6.Axis.PlcToNc <-> Inputs/FromPlc
//   lfe_motion Instance <-> NC-Task 1 SAF/Axes/Axis 7
//     PlcTask Inputs/Main.M7.Axis.NcToPlc <-> Outputs/ToPlc
//     PlcTask Outputs/Main.M7.Axis.PlcToNc <-> Inputs/FromPlc
//   lfe_motion Instance <-> NC-Task 1 SAF/Axes/Axis 8
//     PlcTask Inputs/Main.M8.Axis.NcToPlc <-> Outputs/ToPlc
//     PlcTask Outputs/Main.M8.Axis.PlcToNc <-> Inputs/FromPlc
//   lfe_motion Instance <-> NC-Task 1 SAF/Axes/Axis 9
//     PlcTask Inputs/Main.M9.Axis.NcToPlc <-> Outputs/ToPlc
//     PlcTask Outputs/Main.M9.Axis.PlcToNc <-> Inputs/FromPlc
//   lfe_motion Instance <-> NC-Task 1 SAF/Axes/DIODE HORIZ X
//     PlcTask Inputs/Main.M53.Axis.NcToPlc <-> Outputs/ToPlc
//     PlcTask Outputs/Main.M53.Axis.PlcToNc <-> Inputs/FromPlc
//   lfe_motion Instance <-> NC-Task 1 SAF/Axes/DIODE VERT Y
//     PlcTask Inputs/Main.M54.Axis.NcToPlc <-> Outputs/ToPlc
//     PlcTask Outputs/Main.M54.Axis.PlcToNc <-> Inputs/FromPlc
//   lfe_motion Instance <-> NC-Task 1 SAF/Axes/EM3L0-X-M55
//     PlcTask Inputs/Main.M55.Axis.NcToPlc <-> Outputs/ToPlc
//     PlcTask Outputs/Main.M55.Axis.PlcToNc <-> Inputs/FromPlc
//   lfe_motion Instance <-> NC-Task 1 SAF/Axes/EM3L0-Y-M56
//     PlcTask Inputs/Main.M56.Axis.NcToPlc <-> Outputs/ToPlc
//     PlcTask Outputs/Main.M56.Axis.PlcToNc <-> Inputs/FromPlc
//   lfe_motion Instance <-> NC-Task 1 SAF/Axes/PF1L0-WFS-MMS-01
//     PlcTask Inputs/Main.M31.Axis.NcToPlc <-> Outputs/ToPlc
//     PlcTask Outputs/Main.M31.Axis.PlcToNc <-> Inputs/FromPlc
//   lfe_motion Instance <-> NC-Task 1 SAF/Axes/PF1L0-WFS-MMS-02
//     PlcTask Inputs/Main.M32.Axis.NcToPlc <-> Outputs/ToPlc
//     PlcTask Outputs/Main.M32.Axis.PlcToNc <-> Inputs/FromPlc
//   lfe_motion Instance <-> NC-Task 1 SAF/Axes/RETICLE HORIZ X
//     PlcTask Inputs/Main.M51.Axis.NcToPlc <-> Outputs/ToPlc
//     PlcTask Outputs/Main.M51.Axis.PlcToNc <-> Inputs/FromPlc
//   lfe_motion Instance <-> NC-Task 1 SAF/Axes/RETICLE VERT Y
//     PlcTask Inputs/Main.M52.Axis.NcToPlc <-> Outputs/ToPlc
//     PlcTask Outputs/Main.M52.Axis.PlcToNc <-> Inputs/FromPlc
//   lfe_motion Instance <-> NC-Task 1 SAF/Axes/SL1L0-BOTTOM-M41
//     PlcTask Inputs/Main.M41.Axis.NcToPlc <-> Outputs/ToPlc
//     PlcTask Outputs/Main.M41.Axis.PlcToNc <-> Inputs/FromPlc
//   lfe_motion Instance <-> NC-Task 1 SAF/Axes/SL1L0-NORTH-M44
//     PlcTask Inputs/Main.M44.Axis.NcToPlc <-> Outputs/ToPlc
//     PlcTask Outputs/Main.M44.Axis.PlcToNc <-> Inputs/FromPlc
//   lfe_motion Instance <-> NC-Task 1 SAF/Axes/SL1L0-SOUTH-M42
//     PlcTask Inputs/Main.M42.Axis.NcToPlc <-> Outputs/ToPlc
//     PlcTask Outputs/Main.M42.Axis.PlcToNc <-> Inputs/FromPlc
//   lfe_motion Instance <-> NC-Task 1 SAF/Axes/SL1L0-TOP-M43
//     PlcTask Inputs/Main.M43.Axis.NcToPlc <-> Outputs/ToPlc
//     PlcTask Outputs/Main.M43.Axis.PlcToNc <-> Inputs/FromPlc
//   lfe_motion Instance <-> NC-Task 1 SAF/Axes/SL2L0-BOTTOM-M45
//     PlcTask Inputs/Main.M45.Axis.NcToPlc <-> Outputs/ToPlc
//     PlcTask Outputs/Main.M45.Axis.PlcToNc <-> Inputs/FromPlc
//   lfe_motion Instance <-> NC-Task 1 SAF/Axes/SL2L0-NORTH-M48
//     PlcTask Inputs/Main.M48.Axis.NcToPlc <-> Outputs/ToPlc
//     PlcTask Outputs/Main.M48.Axis.PlcToNc <-> Inputs/FromPlc
//   lfe_motion Instance <-> NC-Task 1 SAF/Axes/SL2L0-SOUTH-M46
//     PlcTask Inputs/Main.M46.Axis.NcToPlc <-> Outputs/ToPlc
//     PlcTask Outputs/Main.M46.Axis.PlcToNc <-> Inputs/FromPlc
//   lfe_motion Instance <-> NC-Task 1 SAF/Axes/SL2L0-TOP-M47
//     PlcTask Inputs/Main.M47.Axis.NcToPlc <-> Outputs/ToPlc
//     PlcTask Outputs/Main.M47.Axis.PlcToNc <-> Inputs/FromPlc
//   lfe_motion Instance <-> NC-Task 1 SAF/Axes/SL3L0-BOTTOM-M59
//     PlcTask Inputs/Main.M59.Axis.NcToPlc <-> Outputs/ToPlc
//     PlcTask Outputs/Main.M59.Axis.PlcToNc <-> Inputs/FromPlc
//   lfe_motion Instance <-> NC-Task 1 SAF/Axes/SL3L0-NORTH-M62
//     PlcTask Inputs/Main.M62.Axis.NcToPlc <-> Outputs/ToPlc
//     PlcTask Outputs/Main.M62.Axis.PlcToNc <-> Inputs/FromPlc
//   lfe_motion Instance <-> NC-Task 1 SAF/Axes/SL3L0-SOUTH-M61
//     PlcTask Inputs/Main.M61.Axis.NcToPlc <-> Outputs/ToPlc
//     PlcTask Outputs/Main.M61.Axis.PlcToNc <-> Inputs/FromPlc
//   lfe_motion Instance <-> NC-Task 1 SAF/Axes/SL3L0-TOP-M60
//     PlcTask Inputs/Main.M60.Axis.NcToPlc <-> Outputs/ToPlc
//     PlcTask Outputs/Main.M60.Axis.PlcToNc <-> Inputs/FromPlc
//   lfe_motion Instance <-> NC-Task 1 SAF/Axes/XTAL ANGLE X
//     PlcTask Inputs/Main.M49.Axis.NcToPlc <-> Outputs/ToPlc
//     PlcTask Outputs/Main.M49.Axis.PlcToNc <-> Inputs/FromPlc
//   lfe_motion Instance <-> NC-Task 1 SAF/Axes/XTAL VERT Y
//     PlcTask Inputs/Main.M50.Axis.NcToPlc <-> Outputs/ToPlc
//     PlcTask Outputs/Main.M50.Axis.PlcToNc <-> Inputs/FromPlc

CONFIGURATION lfe_motion
    RESOURCE PLC ON TwinCAT3
        TASK PlcTask(INTERVAL := T#10ms, PRIORITY := 20);
        PROGRAM PRG_1_PlcTask WITH PlcTask : PRG_1_PlcTask;
    END_RESOURCE
END_CONFIGURATION

// ---- GVLs/GVL.TcGVL
{attribute 'qualified_only'}
VAR_GLOBAL
    {attribute 'pytmc' := 'pv: PLC:LFE:MOTION:ARB:01'}
    fbArbiter: FB_Arbiter(1);

    {attribute 'pytmc' := 'pv: PLC:LFE:MOTION:ARB:02'}
    fbArbiter2: FB_Arbiter(2);

    {attribute 'pytmc' := 'pv: PLC:LFE:MOTION:FFO:01'}
    {attribute 'TcLinkTo' := '.q_xFastFaultOut:=TIIB[PMPS_FFO]^Channel 1^Output'}
    fbFastFaultOutput1: FB_HardwareFFOutput := (bAutoReset := TRUE, i_sNetID := '172.21.88.66.1.1');
	{attribute 'pytmc' := 'pv: PLC:LFE:MOTION:FFO:02'}
	fbFastFaultOutput1a: FB_HardwareFFOutput := (bAutoReset := TRUE, i_sNetID := '172.21.88.66.1.1');
	{attribute 'pytmc' := 'pv: PLC:LFE:MOTION:FFO:03'}
	fbFastFaultOutput1b: FB_HardwareFFOutput := (bAutoReset := TRUE, i_sNetID := '172.21.88.66.1.1');
	{attribute 'pytmc' := 'pv: PLC:LFE:MOTION:FFO:04'}
	fbFastFaultOutput1c: FB_HardwareFFOutput := (bAutoReset := TRUE, i_sNetID := '172.21.88.66.1.1');
	{attribute 'pytmc' := 'pv: PLC:LFE:MOTION:FFO:05'}
	fbFastFaultOutput1d: FB_HardwareFFOutput := (bAutoReset := TRUE, i_sNetID := '172.21.88.66.1.1');
    {attribute 'pytmc' := 'pv: PLC:LFE:MOTION:FFO:06'}
    {attribute 'TcLinkTo' := '.q_xFastFaultOut:=TIIB[PMPS_FFO]^Channel 2^Output'}
    fbFastFaultOutput2: FB_HardwareFFOutput := (bAutoReset := TRUE, i_sNetID := '172.21.88.66.1.1');

    {attribute 'pytmc' := 'pv: PLC:LFE:MOTION:PMPS:ReqTrans'}
    rReqTrans AT %I*		: ARRAY [1..PMPS_GVL.AUX_ATTENUATORS] OF ST_PMPS_Attenuator_IO;
    {attribute 'pytmc' := 'pv: PLC:LFE:MOTION:PMPS:CurTrans'}
    rCurTrans AT %Q*		: ARRAY [1..PMPS_GVL.AUX_ATTENUATORS] OF ST_PMPS_Attenuator_IO;

    ePF1L0State: E_WFS_States;
END_VAR

// ---- GVLs/Main.TcGVL
{attribute 'qualified_only'}
VAR_GLOBAL
(*
    Only includes motor definitions for the IOC
    These are hard-coded to be Main.M#,
    but are very convenient to store in a GVL,
    hence the confusing namespace here

    This should be refactored once the IOC
    supports arbitrary ads paths for motors
*)
    // AT2L0-SOLID: 19 Axes
    {attribute 'pytmc' := 'pv: AT2L0:XTES:MMS:01'}
    {attribute 'TcLinkTo' := '.bLimitForwardEnable  := TIIB[AT2L0-EL7041-01]^STM Status^Status^Digital input 2;
                              .bLimitBackwardEnable := TIIB[AT2L0-EL7041-01]^STM Status^Status^Digital input 1
    '}
    M1: ST_MotionStage := (sName := 'AT2L0:XTES:MMS:01');
    {attribute 'pytmc' := 'pv: AT2L0:XTES:MMS:02'}
    {attribute 'TcLinkTo' := '.bLimitForwardEnable  := TIIB[AT2L0-EL7041-02]^STM Status^Status^Digital input 2;
                              .bLimitBackwardEnable := TIIB[AT2L0-EL7041-02]^STM Status^Status^Digital input 1
    '}
    M2: ST_MotionStage := (sName := 'AT2L0:XTES:MMS:02');
    {attribute 'pytmc' := 'pv: AT2L0:XTES:MMS:03'}
    {attribute 'TcLinkTo' := '.bLimitForwardEnable  := TIIB[AT2L0-EL7041-03]^STM Status^Status^Digital input 2;
                              .bLimitBackwardEnable := TIIB[AT2L0-EL7041-03]^STM Status^Status^Digital input 1
    '}
    M3: ST_MotionStage := (sName := 'AT2L0:XTES:MMS:03');
    {attribute 'pytmc' := 'pv: AT2L0:XTES:MMS:04'}
    {attribute 'TcLinkTo' := '.bLimitForwardEnable  := TIIB[AT2L0-EL7041-04]^STM Status^Status^Digital input 2;
                              .bLimitBackwardEnable := TIIB[AT2L0-EL7041-04]^STM Status^Status^Digital input 1
    '}
    M4: ST_MotionStage := (sName := 'AT2L0:XTES:MMS:04');
    {attribute 'pytmc' := 'pv: AT2L0:XTES:MMS:05'}
    {attribute 'TcLinkTo' := '.bLimitForwardEnable  := TIIB[AT2L0-EL7041-05]^STM Status^Status^Digital input 2;
                              .bLimitBackwardEnable := TIIB[AT2L0-EL7041-05]^STM Status^Status^Digital input 1
    '}
    M5: ST_MotionStage := (sName := 'AT2L0:XTES:MMS:05');
    {attribute 'pytmc' := 'pv: AT2L0:XTES:MMS:06'}
    {attribute 'TcLinkTo' := '.bLimitForwardEnable  := TIIB[AT2L0-EL7041-06]^STM Status^Status^Digital input 2;
                              .bLimitBackwardEnable := TIIB[AT2L0-EL7041-06]^STM Status^Status^Digital input 1
    '}
    M6: ST_MotionStage := (sName := 'AT2L0:XTES:MMS:06');
    {attribute 'pytmc' := 'pv: AT2L0:XTES:MMS:07'}
    {attribute 'TcLinkTo' := '.bLimitForwardEnable  := TIIB[AT2L0-EL7041-07]^STM Status^Status^Digital input 2;
                              .bLimitBackwardEnable := TIIB[AT2L0-EL7041-07]^STM Status^Status^Digital input 1
    '}
    M7: ST_MotionStage := (sName := 'AT2L0:XTES:MMS:07');
    {attribute 'pytmc' := 'pv: AT2L0:XTES:MMS:08'}
    {attribute 'TcLinkTo' := '.bLimitForwardEnable  := TIIB[AT2L0-EL7041-08]^STM Status^Status^Digital input 2;
                              .bLimitBackwardEnable := TIIB[AT2L0-EL7041-08]^STM Status^Status^Digital input 1
    '}
    M8: ST_MotionStage := (sName := 'AT2L0:XTES:MMS:08');
    {attribute 'pytmc' := 'pv: AT2L0:XTES:MMS:09'}
    {attribute 'TcLinkTo' := '.bLimitForwardEnable  := TIIB[AT2L0-EL7041-09]^STM Status^Status^Digital input 2;
                              .bLimitBackwardEnable := TIIB[AT2L0-EL7041-09]^STM Status^Status^Digital input 1
    '}
    M9: ST_MotionStage := (sName := 'AT2L0:XTES:MMS:09');
    {attribute 'pytmc' := 'pv: AT2L0:XTES:MMS:10'}
    {attribute 'TcLinkTo' := '.bLimitForwardEnable  := TIIB[AT2L0-EL7041-10]^STM Status^Status^Digital input 2;
                              .bLimitBackwardEnable := TIIB[AT2L0-EL7041-10]^STM Status^Status^Digital input 1
    '}
    M10: ST_MotionStage := (sName := 'AT2L0:XTES:MMS:10');
    {attribute 'pytmc' := 'pv: AT2L0:XTES:MMS:11'}
    {attribute 'TcLinkTo' := '.bLimitForwardEnable  := TIIB[AT2L0-EL7041-11]^STM Status^Status^Digital input 2;
                              .bLimitBackwardEnable := TIIB[AT2L0-EL7041-11]^STM Status^Status^Digital input 1
    '}
    M11: ST_MotionStage := (sName := 'AT2L0:XTES:MMS:11');
    {attribute 'pytmc' := 'pv: AT2L0:XTES:MMS:12'}
    {attribute 'TcLinkTo' := '.bLimitForwardEnable  := TIIB[AT2L0-EL7041-12]^STM Status^Status^Digital input 2;
                              .bLimitBackwardEnable := TIIB[AT2L0-EL7041-12]^STM Status^Status^Digital input 1
    '}
    M12: ST_MotionStage := (sName := 'AT2L0:XTES:MMS:12');
    {attribute 'pytmc' := 'pv: AT2L0:XTES:MMS:13'}
    {attribute 'TcLinkTo' := '.bLimitForwardEnable  := TIIB[AT2L0-EL7041-13]^STM Status^Status^Digital input 2;
                              .bLimitBackwardEnable := TIIB[AT2L0-EL7041-13]^STM Status^Status^Digital input 1
    '}
    M13: ST_MotionStage := (sName := 'AT2L0:XTES:MMS:13');
    {attribute 'pytmc' := 'pv: AT2L0:XTES:MMS:14'}
    {attribute 'TcLinkTo' := '.bLimitForwardEnable  := TIIB[AT2L0-EL7041-14]^STM Status^Status^Digital input 2;
                              .bLimitBackwardEnable := TIIB[AT2L0-EL7041-14]^STM Status^Status^Digital input 1
    '}
    M14: ST_MotionStage := (sName := 'AT2L0:XTES:MMS:14');
    {attribute 'pytmc' := 'pv: AT2L0:XTES:MMS:15'}
    {attribute 'TcLinkTo' := '.bLimitForwardEnable  := TIIB[AT2L0-EL7041-15]^STM Status^Status^Digital input 2;
                              .bLimitBackwardEnable := TIIB[AT2L0-EL7041-15]^STM Status^Status^Digital input 1
    '}
    M15: ST_MotionStage := (sName := 'AT2L0:XTES:MMS:15');
    {attribute 'pytmc' := 'pv: AT2L0:XTES:MMS:16'}
    {attribute 'TcLinkTo' := '.bLimitForwardEnable  := TIIB[AT2L0-EL7041-16]^STM Status^Status^Digital input 2;
                              .bLimitBackwardEnable := TIIB[AT2L0-EL7041-16]^STM Status^Status^Digital input 1
    '}
    M16: ST_MotionStage := (sName := 'AT2L0:XTES:MMS:16');
    {attribute 'pytmc' := 'pv: AT2L0:XTES:MMS:17'}
    {attribute 'TcLinkTo' := '.bLimitForwardEnable  := TIIB[AT2L0-EL7041-17]^STM Status^Status^Digital input 2;
                              .bLimitBackwardEnable := TIIB[AT2L0-EL7041-17]^STM Status^Status^Digital input 1
    '}
    M17: ST_MotionStage := (sName := 'AT2L0:XTES:MMS:17');
    {attribute 'pytmc' := 'pv: AT2L0:XTES:MMS:18'}
    {attribute 'TcLinkTo' := '.bLimitForwardEnable  := TIIB[AT2L0-EL7041-18]^STM Status^Status^Digital input 2;
                              .bLimitBackwardEnable := TIIB[AT2L0-EL7041-18]^STM Status^Status^Digital input 1
    '}
    M18: ST_MotionStage := (sName := 'AT2L0:XTES:MMS:18');
    {attribute 'pytmc' := 'pv: AT2L0:XTES:MMS:19'}
    {attribute 'TcLinkTo' := '.bLimitForwardEnable  := TIIB[AT2L0-EL7041-19]^STM Status^Status^Digital input 2;
                              .bLimitBackwardEnable := TIIB[AT2L0-EL7041-19]^STM Status^Status^Digital input 1
    '}
    M19: ST_MotionStage := (sName := 'AT2L0:XTES:MMS:19');

    // IM1L0-XTES: 3 Axes
    {attribute 'pytmc' := 'pv: IM1L0:XTES:MMS'}
    {attribute 'TcLinkTo' := '.bLimitForwardEnable  := TIIB[IM1L0-EL7041]^STM Status^Status^Digital input 1;
                              .bBrakeRelease        := TIIB[IM1L0-EL2004]^Channel 1^Output'}
    M20: ST_MotionStage := (sName := 'IM1L0:XTES:MMS');
    {attribute 'pytmc' := 'pv: IM1L0:XTES:CLZ'}
    {attribute 'TcLinkTo' := '.bHome := TIIB[IM1L0-EL1088]^Channel 2^Input'}
    M21: ST_MotionStage := (sName := 'IM1L0:XTES:CLZ');
    {attribute 'pytmc' := 'pv: IM1L0:XTES:CLF'}
    {attribute 'TcLinkTo' := '.bHome := TIIB[IM1L0-EL1088]^Channel 4^Input'}
    M22: ST_MotionStage := (sName := 'IM1L0:XTES:CLF');

    // IM1L1-PPM: 1 Axis
    {attribute 'pytmc' := 'pv: IM1L1:PPM:MMS'}
    {attribute 'TcLinkTo' := '.bLimitForwardEnable  := TIIB[IM1L1-EL7041]^STM Status^Status^Digital input 1;
                              .bLimitBackwardEnable := TIIB[IM1L1-EL7041]^STM Status^Status^Digital input 2;
                              .bBrakeRelease        := TIIB[IM1L1-EL2004]^Channel 1^Output'}
    M23: ST_MotionStage := (sName := 'IM1L1:PPM:MMS');

    // IM2L0-XTES: 3 Axes
    {attribute 'pytmc' := 'pv: IM2L0:XTES:MMS'}
    {attribute 'TcLinkTo' := '.bBrakeRelease        := TIIB[IM2L0-EL2004]^Channel 1^Output'}
    M24: ST_MotionStage := (sName := 'IM2L0:XTES:MMS');
    {attribute 'pytmc' := 'pv: IM2L0:XTES:CLZ'}
    {attribute 'TcLinkTo' := '.bHome := TIIB[IM2L0-EL1088]^Channel 2^Input'}
    M25: ST_MotionStage := (sName := 'IM2L0:XTES:CLZ');
    {attribute 'pytmc' := 'pv: IM2L0:XTES:CLF'}
    {attribute 'TcLinkTo' := '.bHome := TIIB[IM2L0-EL1088]^Channel 4^Input'}
    M26: ST_MotionStage := (sName := 'IM2L0:XTES:CLF');

    // IM3L0-PPM: 1 Axes
    {attribute 'pytmc' := 'pv: IM3L0:PPM:MMS'}
    {attribute 'TcLinkTo' := '.bLimitForwardEnable  := TIIB[IM3L0-EL7041]^STM Status^Status^Digital input 1;
                              .bLimitBackwardEnable := TIIB[IM3L0-EL7041]^STM Status^Status^Digital input 2;
                              .bBrakeRelease        := TIIB[IM3L0-EL2004]^Channel 1^Output'}
    M27: ST_MotionStage := (sName := 'IM3L0:PPM:MMS');

    // IM4L0-XTES: 3 Axes
    {attribute 'pytmc' := 'pv: IM4L0:XTES:MMS'}

    {attribute 'TcLinkTo' := '.bLimitForwardEnable  := TIIB[IM4L0-EL7041]^STM Status^Status^Digital input 1;
                              .bBrakeRelease        := TIIB[IM4L0-EL2004]^Channel 1^Output'}
    M28: ST_MotionStage := (sName := 'IM4L0:XTES:MMS');
    {attribute 'pytmc' := 'pv: IM4L0:XTES:CLZ'}
    {attribute 'TcLinkTo' := '.bHome := TIIB[IM4L0-EL1088]^Channel 2^Input'}
    M29: ST_MotionStage := (sName := 'IM4L0:XTES:CLZ');
    {attribute 'pytmc' := 'pv: IM4L0:XTES:CLF'}
    {attribute 'TcLinkTo' := '.bHome := TIIB[IM4L0-EL1088]^Channel 4^Input'}
    M30: ST_MotionStage := (sName := 'IM4L0:XTES:CLF');

    // PF1L0-WFS: 2 Axes
    {attribute 'pytmc' := 'pv: PF1L0:WFS:MMS:Y'}
    {attribute 'TcLinkTo' := '.bLimitForwardEnable  := TIIB[PF1L0-EL7041-01]^STM Status^Status^Digital input 1;
                              .bLimitBackwardEnable := TIIB[PF1L0-EL7041-01]^STM Status^Status^Digital input 2;
                              .bBrakeRelease        := TIIB[PF1L0-EL2004]^Channel 1^Output;
                              .nRawEncoderULINT     := TIIB[PF1L0-EL5042]^FB Inputs Channel 2^Position'}
    M31: ST_MotionStage := (sName := 'PF1L0:WFS:MMS:01');
    {attribute 'pytmc' := 'pv: PF1L0:WFS:MMS:Z'}
    {attribute 'TcLinkTo' := '.nRawEncoderULINT     := TIIB[PF1L0-EL5042]^FB Inputs Channel 1^Position'}
    M32: ST_MotionStage := (sName := 'PF1L0:WFS:MMS:02');

    // RTDSL0: 8 Axes
    {attribute 'pytmc' := 'pv: RTDSL0:DIODE:MMS:01'}
    {attribute 'TcLinkTo' := '.bLimitForwardEnable  := TIIB[RTDSL0-EL7041-01]^STM Status^Status^Digital input 1;
                              .bLimitBackwardEnable := TIIB[RTDSL0-EL7041-01]^STM Status^Status^Digital input 2'}
    M33: ST_MotionStage := (sName := 'RTDSL0:DIODE:MMS:01');
    M34: ST_MotionStage;
    M35: ST_MotionStage;
    M36: ST_MotionStage;
    M37: ST_MotionStage;
    //to be uncommented when the mccallister stage on RTDSK0 is moved to RTDSLo
    (*
    {attribute 'pytmc' := 'pv: RTDSL0:SCRP:MMS:01'}
    {attribute 'TcLinkTo' := '.bLimitForwardEnable  := TIIB[RTDSL0-EL7041-02]^STM Status^Status^Digital input 1;
                              .bLimitBackwardEnable := TIIB[RTDSL0-EL7041-02]^STM Status^Status^Digital input 2'}
    M34: ST_MotionStage := (sName := 'RTDSL0:SCRP:MMS:01');
    {attribute 'pytmc' := 'pv: RTDSL0:SCRP:MMS:02'}
    {attribute 'TcLinkTo' := '.bLimitForwardEnable  := TIIB[RTDSL0-EL7041-03]^STM Status^Status^Digital input 1;
                              .bLimitBackwardEnable := TIIB[RTDSL0-EL7041-03]^STM Status^Status^Digital input 2'}
    M35: ST_MotionStage := (sName := 'RTDSL0:SCRP:MMS:02');
    {attribute 'pytmc' := 'pv: RTDSL0:SCRP:MMS:03'}
    {attribute 'TcLinkTo' := '.bLimitForwardEnable  := TIIB[RTDSL0-EL7041-04]^STM Status^Status^Digital input 1;
                              .bLimitBackwardEnable := TIIB[RTDSL0-EL7041-04]^STM Status^Status^Digital input 2'}
    M36: ST_MotionStage := (sName := 'RTDSL0:SCRP:MMS:03');
    *)
    //LDM on RTDSL0
    {attribute 'pytmc' := 'pv: RTDSL0:LDM:MMS:01'}
    {attribute 'TcLinkTo' := '.bLimitForwardEnable  := TIIB[RTDSL0-EL7041-05]^STM Status^Status^Digital input 1;
                              .bLimitBackwardEnable := TIIB[RTDSL0-EL7041-05]^STM Status^Status^Digital input 2;
                               .nRawEncoderINT := TIIB[Term 113 (EL3054)]^AI Standard Channel 1^Value'}
    //M37: ST_MotionStage := (sName := 'RTDSL0:LDM:MMS:01');
    M38: ST_MotionStage;
    M39: ST_MotionStage;
    M40: ST_MotionStage;

    // to be uncommented when mccallister stage is moved from RTDSK0 -> RTDSL0
    (*
    {attribute 'pytmc' := 'pv: RTDSL0:SCRP:LED:01'}
    {attribute 'TcLinkTo' := '.bLimitForwardEnable  := TIIB[RTDSK0-EL7041-04]^STM Status^Status^Digital input 1;
                              .bLimitBackwardEnable := TIIB[RTDSK0-EL7041-04]^STM Status^Status^Digital input 2'}
    LED1: ENUM_XPIM_States;
    *)


    // SL1L0-POWER: 4 Axes
    {attribute 'pytmc' := 'pv: SL1L0:POWER:MMS:BOTTOM'}
    {attribute 'TcLinkTo' := '.bLimitForwardEnable  := TIIB[SL1L0-EL7041-E1]^STM Status^Status^Digital input 2;
                              .bLimitBackwardEnable := TIIB[SL1L0-EL7041-E1]^STM Status^Status^Digital input 1'}
    M41: ST_MotionStage := (sName := 'SL1L0:POWER:MMS:BOTTOM');
        {attribute 'pytmc' := 'pv: SL1L0:POWER:MMS:SOUTH'}
    {attribute 'TcLinkTo' := '.bLimitForwardEnable  := TIIB[SL1L0-EL7041-E3]^STM Status^Status^Digital input 1;
                              .bLimitBackwardEnable := TIIB[SL1L0-EL7041-E3]^STM Status^Status^Digital input 2'}
    M42: ST_MotionStage := (sName := 'SL1L0:POWER:MMS:SOUTH');
    {attribute 'pytmc' := 'pv: SL1L0:POWER:MMS:TOP'}
    {attribute 'TcLinkTo' := '.bLimitForwardEnable  := TIIB[SL1L0-EL7041-E5]^STM Status^Status^Digital input 2;
                              .bLimitBackwardEnable := TIIB[SL1L0-EL7041-E5]^STM Status^Status^Digital input 1'}
    M43: ST_MotionStage := (sName := 'SL1L0:POWER:MMS:TOP');
    {attribute 'pytmc' := 'pv: SL1L0:POWER:MMS:NORTH'}
    {attribute 'TcLinkTo' := '.bLimitForwardEnable  := TIIB[SL1L0-EL7041-E7]^STM Status^Status^Digital input 1;
                              .bLimitBackwardEnable := TIIB[SL1L0-EL7041-E7]^STM Status^Status^Digital input 2'}
    M44: ST_MotionStage := (sName := 'SL1L0:POWER:MMS:NORTH');

    // SL2L0-POWER: 4 Axes
    {attribute 'pytmc' := 'pv: SL2L0:POWER:MMS:BOTTOM'}
    {attribute 'TcLinkTo' := '.bLimitForwardEnable  := TIIB[SL2L0-EL7041-E1]^STM Status^Status^Digital input 2;
                              .bLimitBackwardEnable := TIIB[SL2L0-EL7041-E1]^STM Status^Status^Digital input 1'}
    M45: ST_MotionStage := (sName := 'SL2L0:POWER:MMS:BOTTOM');
    {attribute 'pytmc' := 'pv: SL2L0:POWER:MMS:SOUTH'}
    {attribute 'TcLinkTo' := '.bLimitForwardEnable  := TIIB[SL2L0-EL7041-E3]^STM Status^Status^Digital input 1;
                              .bLimitBackwardEnable := TIIB[SL2L0-EL7041-E3]^STM Status^Status^Digital input 2'}
    M46: ST_MotionStage := (sName := 'SL2L0:POWER:MMS:SOUTH');
    {attribute 'pytmc' := 'pv: SL2L0:POWER:MMS:TOP'}
    {attribute 'TcLinkTo' := '.bLimitForwardEnable  := TIIB[SL2L0-EL7041-E5]^STM Status^Status^Digital input 2;
                              .bLimitBackwardEnable := TIIB[SL2L0-EL7041-E5]^STM Status^Status^Digital input 1'}
    M47: ST_MotionStage := (sName := 'SL2L0:POWER:MMS:TOP');
    {attribute 'pytmc' := 'pv: SL2L0:POWER:MMS:NORTH'}
    {attribute 'TcLinkTo' := '.bLimitForwardEnable  := TIIB[SL2L0-EL7041-E7]^STM Status^Status^Digital input 1;
                              .bLimitBackwardEnable := TIIB[SL2L0-EL7041-E7]^STM Status^Status^Digital input 2'}
    M48: ST_MotionStage := (sName := 'SL2L0:POWER:MMS:NORTH');

    // SP1L0-KMONO: 6 Axes
    {attribute 'pytmc' := 'pv: SP1L0:KMONO:MMS:XTAL_ANGLE'}
    M49: ST_MotionStage := (sName := 'SP1L0:KMONO:MMS:XTAL_ANGLE');
    {attribute 'pytmc' := 'pv: SP1L0:KMONO:MMS:XTAL_VERT'}
    //{attribute 'TcLinkTo' := '.bLimitForwardEnable  := TIIB[SP1L0-EL7041-E2-MOTORS]^STM Status^Status^Digital input 2;
    //                          .bLimitBackwardEnable := TIIB[SP1L0-EL7041-E2-MOTORS]^STM Status^Status^Digital input 1'}
    M50: ST_MotionStage := (sName := 'SP1L0:KMONO:MMS:XTAL_VERT');
    {attribute 'pytmc' := 'pv: SP1L0:KMONO:MMS:RET_HORIZ'}
    //{attribute 'TcLinkTo' := '.bLimitForwardEnable  := TIIB[SP1L0-EL7041-E3-MOTORS]^STM Status^Status^Digital input 2;
    //                          .bLimitBackwardEnable := TIIB[SP1L0-EL7041-E3-MOTORS]^STM Status^Status^Digital input 1'}
    M51: ST_MotionStage := (sName := 'SP1L0:KMONO:MMS:RET_HORIZ');
    {attribute 'pytmc' := 'pv: SP1L0:KMONO:MMS:RET_VERT'}
    //{attribute 'TcLinkTo' := '.bLimitForwardEnable  := TIIB[SP1L0-EL7041-E4-MOTORS]^STM Status^Status^Digital input 1;
    //                          .bLimitBackwardEnable := TIIB[SP1L0-EL7041-E4-MOTORS]^STM Status^Status^Digital input 2'}
    M52: ST_MotionStage := (sName := 'SP1L0:KMONO:MMS:RET_VERT');
    {attribute 'pytmc' := 'pv: SP1L0:KMONO:MMS:DIODE_HORIZ'}
    //{attribute 'TcLinkTo' := '.bLimitForwardEnable  := TIIB[SP1L0-EL7041-E5-MOTORS]^STM Status^Status^Digital input 2;
    //                          .bLimitBackwardEnable := TIIB[SP1L0-EL7041-E5-MOTORS]^STM Status^Status^Digital input 1'}
    M53: ST_MotionStage := (sName := 'SP1L0:KMONO:MMS:DIODE_HORIZ');
    {attribute 'pytmc' := 'pv: SP1L0:KMONO:MMS:DIODE_VERT'}
    //{attribute 'TcLinkTo' := '.bLimitForwardEnable  := TIIB[SP1L0-EL7041-E6-MOTORS]^STM Status^Status^Digital input 1;
    //                          .bLimitBackwardEnable := TIIB[SP1L0-EL7041-E6-MOTORS]^STM Status^Status^Digital input 2'}
    M54: ST_MotionStage := (sName := 'SP1L0:KMONO:MMS:DIODE_VERT');

        // Three_Stage_RTDSX0: 3 Axes
     (*   to uncomment when stage is moved to RTDSL0
    {attribute 'pytmc' := 'pv: RTDSX0:MMS:01'}
    {attribute 'TcLinkTo' := '.bLimitForwardEnable  := TIIB[SP1L0-EL7041-E2-MOTORS]^STM Status^Status^Digital input 2;
                              .bLimitBackwardEnable := TIIB[SP1L0-EL7041-E2-MOTORS]^STM Status^Status^Digital input 1'}
    M55: ST_MotionStage := (sName := 'RTDSX0:MMS:01');

     {attribute 'pytmc' := 'pv: RTDSX0:MMS:02'}
    {attribute 'TcLinkTo' := '.bLimitForwardEnable  := TIIB[SP1L0-EL7041-E2-MOTORS]^STM Status^Status^Digital input 2;
                              .bLimitBackwardEnable := TIIB[SP1L0-EL7041-E2-MOTORS]^STM Status^Status^Digital input 1'}
    M56: ST_MotionStage := (sName := 'RTDSX0:MMS:02');

    {attribute 'pytmc' := 'pv: RTDSX0:MMS:03'}
    {attribute 'TcLinkTo' := '.bLimitForwardEnable  := TIIB[SP1L0-EL7041-E2-MOTORS]^STM Status^Status^Digital input 2;
                              .bLimitBackwardEnable := TIIB[SP1L0-EL7041-E2-MOTORS]^STM Status^Status^Digital input 1'}
    M57: ST_MotionStage := (sName := 'RTDSX0:MMS:03');
    *)

    {attribute 'pytmc' := 'pv: EM3L0:IPM:MMS:X'}
    {attribute 'TcLinkTo' := '.nRawEncoderULINT     := TIIB[EM3L0-EL5042-E2]^FB Inputs Channel 1^Position'}
    M55: ST_MotionStage := (sName := 'EM3L0:IPM:MMS:X');
    {attribute 'pytmc' := 'pv: EM3L0:IPM:MMS:Y'}
    {attribute 'TcLinkTo' := '.bBrakeRelease        := TIIB[EM3L0-EL2004-E4]^Channel 1^Output;
                              .nRawEncoderULINT     := TIIB[EM3L0-EL5042-E2]^FB Inputs Channel 2^Position'}
    M56: ST_MotionStage := (sName := 'EM3L0:IPM:MMS:Y');

